IF  OP30_Gripper_RH_Gripper_ctrl.Axis_reference AND OP30_Gripper_RH_Open THEN
	OP30_Gripper_RH_Gripper_ctrl.Position:=OP30_Gripper_Wrk_POS;
	OP30_Gripper_RH_Gripper_ctrl.ABSmove_Start:=TRUE;
	IF OP30_Gripper_RH_Gripper_ctrl.pos_done AND In_range(OP30_Gripper_RH_Gripper_ctrl.Actual_Position,OP30_Gripper_Wrk_POS,1) THEN
		OP30_Gripper_RH_Open:=FALSE;
		OP30_Gripper_RH_Gripper_ctrl.ABSmove_Start:=0;
		OP30_Gripper_RH_State:=1;
	END_IF
END_IF

IF  OP30_Gripper_RH_Gripper_ctrl.Axis_reference AND OP30_Gripper_RH_Close THEN
	OP30_Gripper_RH_Gripper_ctrl.Position:=0;
	OP30_Gripper_RH_Gripper_ctrl.ABSmove_Start:=TRUE;
	IF OP30_Gripper_RH_Gripper_ctrl.pos_done AND In_range(OP30_Gripper_RH_Gripper_ctrl.Actual_Position,0.1,1) THEN
		OP30_Gripper_RH_Close:=FALSE;
		OP30_Gripper_RH_Gripper_ctrl.ABSmove_Start:=0;
		OP30_Gripper_RH_State:=0;
	END_IF	
END_IF

Test(IN:= OP30_Gripper_RH_State AND OP30_Gripper_LH_State , PT:=T#500MS);


OP30_GIUDE_GRP(														// FESTO GUIDE GRIPPER
	bAxis1_Ref_Switch:= , 
	bInit:=  , 
	bErrorReset:= Servo_Reset , 
	bEnable:= Servo_Enable , /// MACHINE ERR REGISTER CHANGE
	bMoveVelocity:= , 
	bHalt:= , 
	bManualMode:=OP30_ManualSelected AND MANUAL_SELECTED , 									//MANUAL REGISTER CHANGE
	fHomePos:= , 
	fOverride:= , 
	fTargetPosition:= OP30_GIUDE_GRP_ctrl.Position, 
	fTargetVelocity:= OP30_GIUDE_GRP_ctrl.Velocity, 
	fAcc:= , 
	fDec:= , 
	Servo_High_Limit:= 100,	
	Servo_Low_Limit:= -100,	 	
	WARNING_LIMIT:= 1,		
	Safe_move_Conditions:= Servo_Safety,
	TORQUE_APPLIED :=  , 					// CHANGE
	Axis:= SR30_GUIDE_GRP_AXIS, 
	bHome:= OP30_GIUDE_GRP_ctrl.Bsethome, 
	bSetPosition:= FESTO_NOT_NEED , 
	bMoveAbsolute:= OP30_GIUDE_GRP_ctrl.ABSmove_Start, 
	bMoveRelative:= NOT_REQ , 
	bMoveTorque:= NOT_REQ , 
	stManualModeAxis:= OP30_GIUDE_GRP_Manual_Axis, 
 	sAxisState=> OP30_GIUDE_GRP_ctrl.Axis_State, 
	baxis_in_home_pos=>OP30_GIUDE_GRP_ctrl.Axis_In_Home ,
	bAxis_ready=> , 
	bAxisInPosition=> , 
	bAxisError=> , 
	bAxisEnabled=> , 
	bAxisHomed=>, 
	bSetPositionDone=> , 
	bHaltDone=> , 
	bSTOPDone=> , 
	bHomeDone=>OP30_GIUDE_GRP_ctrl.Axis_Home_Done , 
	bDone=> , 
	bTorqueReached=> , 
	bsafe_to_move=> , 
	baxis_in_home_pos=> , 
	bABS_Pos_done=> OP30_GIUDE_GRP_ctrl.Axis_In_Pos, 
	Actual_position=>OP30_GIUDE_GRP_ctrl.Actual_Position,
	Actual_velocity=>OP30_GIUDE_GRP_ctrl.Actual_Velocity , 
	Actual_Torque=> );

END_PROGRAM

// ---- POUs/Programs/OP30/OP30_AUTOSEQUENCE.TcPOU
PROGRAM OP30_AUTOSEQUENCE
VAR
	OP30_Oring_OK 	: BOOL;
	FIXTURE_LH		: INT;
	FIXTURE_RH 		: INT;
	del : ton;
	tmp :BOOL;
	Jerk_Check	: TON;
	Gripper_Delay: TON;
	Gripper_Aft_Place_Delay	: TON;
	OP30_STN_MOVER: INT;
	Dry_run : BOOL;
	OP30_Cycle_Time_FB : FB_Cycletime;
	Guide_Control_Temp : BOOL;
	
	PAP_CYC_VAR : BOOL;
	OP30_PAP_Cycle_time : UDINT;
	OP30_Overall_Cyc_Time	: UDINT;
	OP30_PAP_Cycle_Time_FB : FB_Cycletime;
	OP30_Continous_Run : BOOL;
END_VAR

// AUTO MODE
IF (NOT OP30_AutoSelected OR  OP30_ErrorActive OR OP30_HomeRunning ) THEN
	OP30_AutoRunning:= FALSE;
	OP30_AutoSeq:= 10;
END_IF	

IF (NOT OP30_AutoSelected OR  OP30_ErrorActive ) THEN
	OP30_Conveyor_ON:=FALSE;
END_IF	

IF OP30_AutoSelected THEN
	OP30_GIUDE_GRP_ctrl.Position:=OP30_Guide_Pos;
	OP30_GIUDE_GRP_ctrl.Velocity:=50;
	SR30_Vert_servo_ctrl.Velocity:=OP30_HMI_Servo_Speed_Vertical;
	SR30_HORI_servo_ctrl.Velocity:=OP30_HMI_Servo_Speed_Horizontal;	
END_IF

IF NOT OP30_AutoRunning THEN
    OP30_GIUDE_GRP_ctrl.Position:=0;
	OP30_GIUDE_GRP_ctrl.Velocity:=50;
	IF NOT In_Range(OP30_GIUDE_GRP_ctrl.Actual_Position,0,1) THEN
		OP30_GIUDE_GRP_ctrl.ABSmove_Start:=TRUE;
	END_IF	
END_IF

CASE OP30_AutoSeq OF
	    10: IF (OP30_AutoSelected) THEN		// Check Automode Selected
				OP30_AutoSeq:=20;
	        END_IF
		
	    20:IF ( NOT OP30_ErrorActive) THEN		//Check No error
		       OP30_AutoSeq:=30;
      	   END_IF
		   
      	30:IF (NOT OP30_HomeRunning) THEN		//Check No Homerunning
      		   OP30_AutoSeq :=40;
      	   END_IF
		   
        40:IF (OP30_Main.OP30_Modeselection_FB.TempHomeOK)THEN	//Check Machine in Home
      		   OP30_AutoSeq:= 50;
      	   END_IF
		   
      	50:IF ( NOT OP30_OperationCompleted) THEN		// Check Operation Completed Reset
			   OP30_AutoSeq:=60;
      	   END_IF
		   
		60:IF  ( OP30_AutoRunning OR (NOT OP30_AutoRunning AND OP30_HMI_Cycle_Start )) THEN		//Machine Start in Fully Automatic or Press Cycle Start For Semi Automatic
		    OP30_GVL.OP30_HomeConditionOK:=TRUE;
	 			IF( OP30_Main.OP30_Modeselection_FB.HomeConditionOK AND OP30_AutoSelected) THEN
					OP30_GVL.OP30_AutoRunning:=TRUE;
					OP30_GVL.OP30_StepRunning:= FALSE;				
				ELSIF (OP30_Main.OP30_Modeselection_FB.HomeConditionOK AND OP30_StepSelected) THEN
					OP30_GVL.OP30_AutoRunning:=FALSE;
					OP30_GVL.OP30_StepRunning:= TRUE;
				END_IF;
		  END_IF
		   IF ((OP30_AutoRunning OR OP30_StepRunning) AND OP30_StartEnable) THEN
			   	OP30_GIUDE_GRP_ctrl.ABSmove_Start:=TRUE;
				OP30_Conveyor_ON:=TRUE;
				OP30_AutoSeq:= 65;
		   END_IF	
		   
		65 :  OP30_Gripper_LH_Close:=TRUE;  //CHECKING GRIPPER STATE BEFORE GRIPPING
			  OP30_Gripper_RH_Close:=TRUE;
			  IF NOT OP30_Gripper_LH_State AND NOT OP30_Gripper_RH_State THEN
				   OP30_AutoSeq:=66;
			  ELSE 	   
				   OP30_AutoSeq:=220;
			  END_IF 
		   
	    66: PAP_CYC_VAR:=1;
			IF OP30_pick_ready THEN
				OP30_AutoSeq:=70;
			ELSE 
				OP30_AutoSeq:=86;	
			END_IF 
			  
		70 : //MOVING HORIZONTAL SERVO TO PICK POSITION
			  IF (OP30_HORI_SERVO_ON_SFE_WRK OR OP30_HORI_SERVO_ON_HOME OR OP30_HORI_SERVO_ON_WRK_PLACE OR OP30_HORI_SERVO_ON_WRK_PICK )AND OP30_HORI_SERVO_POS_DONE AND NOT SR30_HORI_servo_ctrl.ABSmove_Start THEN 
			   SR30_Hori_servo_ctrl.Position:=OP30_HORI_SERVO_PICK_POS;
               OP30_AutoSeq:=80;
			  END_IF
			 
		80 :  SR30_HORI_servo_ctrl.ABSmove_Start := TRUE;     //HORIZONTAL SERVO MOVING
		       IF OP30_HORI_SERVO_ON_WRK_PICK THEN
				   SR30_HORI_servo_ctrl.ABSmove_Start := FALSE;
				   IF OP30_Gripper_LH_State AND OP30_Gripper_RH_State THEN
				        OP30_AutoSeq:=85;
				   ELSE 
						OP30_AutoSeq:=82;
				   END_IF
			   END_IF
		
	  	82 :  OP30_Gripper_LH_Close:=TRUE;  //CHECKING GRIPPER STATE BEFORE GRIPPING
			  OP30_Gripper_RH_Close:=TRUE;
			  IF NOT OP30_Gripper_LH_State AND NOT OP30_Gripper_RH_State THEN
				   OP30_AutoSeq:=85;
			  END_IF
			   
		85:	   // MOVING VERTICAL SERVO TO PICK POSITION
               IF  OP30_HORI_SERVO_ON_WRK_PICK AND (OP30_VERT_SERVO_ON_SFE_WRK OR OP30_VERT_SERVO_ON_HOME) AND OP30_VERT_SERVO_POS_DONE AND NOT SR30_VERT_servo_ctrl.ABSmove_Start   THEN
				   SR30_Vert_servo_ctrl.Position:=OP30_VERT_SERVO_PICK_POS;
				   SR30_VERT_servo_ctrl.ABSmove_Start := TRUE;
              	   OP30_AutoSeq:=100;			   
			   END_IF
			   
	    86:   IF (OP30_HORI_SERVO_ON_SFE_WRK OR OP30_HORI_SERVO_ON_HOME OR OP30_HORI_SERVO_ON_WRK_PLACE OR OP30_HORI_SERVO_ON_WRK_PICK )AND OP30_HORI_SERVO_POS_DONE AND NOT SR30_HORI_servo_ctrl.ABSmove_Start THEN 
			    SR30_Hori_servo_ctrl.Position:=OP30_HORI_SERVO_SAFE_PICK_POS;
			    SR30_HORI_servo_ctrl.ABSmove_Start := TRUE;
                OP30_AutoSeq:=90;
			  END_IF
  
		90 :   IF OP30_pick_ready THEN  // WAITING FOR O-RING TO BE OK AND THEN MOVING THE VERTICAL SERVO
			 		SR30_Hori_servo_ctrl.Position:=OP30_HORI_SERVO_PICK_POS;
					OP30_AutoSeq:=92;
		       END_IF
			   
		92:  SR30_Hori_servo_ctrl.ABSmove_Start := TRUE;
			 IF OP30_HORI_SERVO_ON_WRK_PICK THEN
				 SR30_Vert_servo_ctrl.Position:=OP30_VERT_SERVO_PICK_POS;
				 SR30_VERT_servo_ctrl.ABSmove_Start := TRUE;
				 OP30_AutoSeq:=100;
			 END_IF
						  						   			   
	   100 : IF OP30_VERT_SERVO_ON_WRK_PICK AND NOT SR30_VERT_servo_ctrl.ABSmove_Start THEN
				 SR30_VERT_servo_ctrl.ABSmove_Start := FALSE;
				 SR30_Vert_servo_ctrl.Position:=OP30_VERT_SERVO_SFE_WRK_POS; // FEEDING SAFE-WORK POSITION TO VERTICAL SERVO
              	 OP30_AutoSeq:=110;			    				   
			 END_IF	   
			   
       110:	IF NOT OP30_Grip_LH_Bypass THEN
				OP30_Gripper_LH_Open:=TRUE; 
			END_IF	
			IF NOT OP30_Grip_RH_Bypass THEN
    			OP30_Gripper_RH_Open:=TRUE;
			END_IF	
			IF Gripper_Delay.Q THEN
				 OP30_AutoSeq:=120;
		    END_IF 
    		
       120: SR30_Hori_servo_ctrl.Position:=(OP30_HORI_SERVO_PICK_POS+OP30_Hori_Ser_Jerk_Pos);
	   		SR30_HORI_servo_ctrl.ABSmove_Start := 1;
			IF Jerk_Check.Q THEN
				OP30_AutoSeq:=130;
			END_IF    
    		   
       130: SR30_VERT_servo_ctrl.ABSmove_Start := TRUE;	   //MOVING VERTICL SERVO TO SAFE-WORK
            IF OP30_VERT_SERVO_ON_SFE_WRK  THEN
    	      SR30_VERT_servo_ctrl.ABSmove_Start := FALSE;
			  OP30_pick_done:=TRUE;
              OP30_AutoSeq:=140;   
    		END_IF
    		   
       140: IF (NOT OP30_Gripper_LH_State AND OP30_Grip_LH_Bypass ) AND OP30_Gripper_RH_State THEN  
    			OP30_AutoSeq:=150;
			ELSIF (NOT OP30_Gripper_RH_State AND OP30_Grip_RH_Bypass) AND OP30_Gripper_LH_State THEN
				OP30_AutoSeq:=150;
			ELSIF OP30_Gripper_LH_State AND OP30_Gripper_RH_State THEN  
    			OP30_AutoSeq:=150;
			ELSIF (NOT OP30_Gripper_LH_State AND NOT OP30_Grip_LH_Bypass) OR (NOT OP30_Gripper_RH_State AND NOT OP30_Grip_RH_Bypass) THEN	
				OP30_AutoSeq:=220;
			ELSIF OP30_Grip_LH_Bypass AND OP30_Grip_RH_Bypass THEN
				OP30_AutoSeq:=250;
			END_IF
    	    		  
       150:  IF OP30_VERT_SERVO_ON_SFE_WRK  THEN // FEEDING PLACE POSITION TO HORIZONTAL SERVO
    		   SR30_Hori_servo_ctrl.Position:=OP30_HORI_SERVO_PLACE_POS;
              OP30_AutoSeq:=160;			 
    		 END_IF
    		   
       160:  SR30_HORI_servo_ctrl.ABSmove_Start := TRUE;    // MOVING HORIZONTAL SERVO TO PLACE POSITION
    		   IF OP30_HORI_SERVO_ON_WRK_PLACE THEN
    			 SR30_HORI_servo_ctrl.ABSmove_Start := FALSE;
    			 OP30_AutoSeq:=170;
    		   END_IF
       
       170: PAP_CYC_VAR:=0;
			IF OP30_HORI_SERVO_ON_WRK_PLACE AND NOT SR30_VERT_servo_ctrl.ABSmove_Start AND OP30_VERT_SERVO_ON_SFE_WRK AND OP30_STN_ENABLE THEN
    	   		SR30_Vert_servo_ctrl.Position:=OP30_VERT_SERVO_PLACE_POS;
              	OP30_AutoSeq:=175;		
      		END_IF
			
	   175: IF FIXTURE_LH<>20 AND FIXTURE_RH<>20 THEN
		   		OP30_AutoSeq:=250;	
			ELSIF FIXTURE_LH<>20 OR FIXTURE_RH<>20 THEN
				OP30_AutoSeq:=260;	
			ELSE
				OP30_AutoSeq:=180;		
	  	    END_IF
    		
       180: SR30_Vert_servo_ctrl.Position:=OP30_VERT_SERVO_PLACE_POS;
			SR30_VERT_servo_ctrl.ABSmove_Start := TRUE; //MOVING VERTICAL SERVO TO PLACE POSITION
    		IF OP30_VERT_SERVO_ON_WRK_PLACE THEN
    			SR30_VERT_servo_ctrl.ABSmove_Start := FALSE;
    		    OP30_AutoSeq:=190;					
    		END_IF	
			
       190: IF FIXTURE_LH=20 AND NOT OP30_Grip_LH_Bypass THEN 
				OP30_Gripper_LH_Close:=TRUE;	
			END_IF	
			IF FIXTURE_RH=20 AND NOT OP30_Grip_RH_Bypass THEN 
				OP30_Gripper_RH_Close:=TRUE;
			END_IF			
			OP30_AutoSeq	:=200;
			OP30_CURR_MOVER	:= OP30_STN_MOVER;
				
	
       200:  //MOVING BACK TO VERTICAL SERVO SAFE POSITION
    		 IF OP30_VERT_SERVO_ON_WRK_PLACE AND NOT SR30_VERT_servo_ctrl.ABSmove_Start THEN
    		   SR30_Vert_servo_ctrl.Position:=OP30_VERT_SERVO_SFE_WRK_POS;
			   IF Gripper_Aft_Place_Delay.Q THEN
                OP30_AutoSeq:=201;
			   END_IF			   
    		 END_IF 
    		 
	   201: IF Dry_Run THEN
				OP30_AutoSeq:=210; 
			END_IF
			IF  FIXTURE_LH=20 AND FIXTURE_RH=20 THEN
				MOVER_CMP_STATUS[OP30_CURR_MOVER][1]:=30 ;
				MOVER_CMP_STATUS[OP30_CURR_MOVER][2]:=30 ;
				OP30_AutoSeq:=210;
			ELSIF FIXTURE_LH=20 THEN
				MOVER_CMP_STATUS[OP30_CURR_MOVER][1]:=30 ;
				OP30_AutoSeq:=210;
			ELSIF FIXTURE_RH=20 THEN
				MOVER_CMP_STATUS[OP30_CURR_MOVER][2]:=30 ;
				OP30_AutoSeq:=210;
			END_IF		 
			 
       210:	   //PROCEEDING FOR NEXT CYCLE 
			  SR30_VERT_servo_ctrl.ABSmove_Start := TRUE;         
              IF OP30_VERT_SERVO_ON_SFE_WRK OR OP30_VERT_SERVO_ON_HOME  THEN
    			SR30_VERT_servo_ctrl.ABSmove_Start := FALSE;			  
				OP30_STN_ENABLE:=0;
				IF OP30_Gripper_LH_State OR OP30_Gripper_RH_State THEN
					OP30_AutoSeq:=220;
				ELSIF (MOVER_CMP_STATUS[OP30_STN_MOVER][1]=30 OR MOVER_CMP_STATUS[OP30_STN_MOVER][2]=30) OR Dry_Run THEN
					STATION_DONE[OP30_CURR_MOVER][OP30_XTS_POS_NO]	:= TRUE;
					IF MOVER_STP_NO[OP30_CURR_MOVER]<>((OP30_XTS_POS_NO*10)+1)THEN
						OP30_AutoSeq:=66;  
					END_IF	
    		  	END_IF  			  
			  END_IF
    		  
       220:  IF (OP30_VERT_SERVO_ON_SFE_WRK OR OP30_VERT_SERVO_ON_HOME OR OP30_VERT_SERVO_ON_WRK_PLACE OR OP30_VERT_SERVO_ON_WRK_PICK) AND NOT SR30_HORI_servo_ctrl.ABSmove_Start AND (OP30_HORI_SERVO_ON_WRK_PLACE OR OP30_HORI_SERVO_ON_WRK_Pick)  THEN
    		   SR30_Hori_servo_ctrl.Position:=OP30_HORI_SERVO_SFE_WRK_POS;
			   SR30_Vert_servo_ctrl.Position:=OP30_VERT_SERVO_SFE_WRK_POS;
               OP30_AutoSeq:=240;			  
    		 END_IF  
    	
       240: SR30_VERT_servo_ctrl.ABSmove_Start := TRUE;	
			IF OP30_VERT_SERVO_ON_SFE_WRK THEN
			 	SR30_HORI_servo_ctrl.ABSmove_Start := TRUE;
             	IF OP30_HORI_SERVO_ON_SFE_WRK THEN
    	  	 	  SR30_HORI_servo_ctrl.ABSmove_Start := FALSE;
      		 	  OP30_Gripper_RH_Close:=TRUE;	
    		 	  OP30_Gripper_LH_Close:=TRUE; 			   
      		 	END_IF
			END_IF	
    		IF NOT OP30_Gripper_LH_State AND NOT OP30_Gripper_RH_State THEN
    		   OP30_AutoSeq:=66;
    		END_IF
			 		
		250://MOVER_CMP_STATUS[OP30_CURR_MOVER][1]:=31;
			//MOVER_CMP_STATUS[OP30_CURR_MOVER][2]:=31;
			OP30_STN_ENABLE:=0;
			IF 	(MOVER_CMP_STATUS[OP30_STN_MOVER][1]=31 AND MOVER_CMP_STATUS[OP30_STN_MOVER][2]=31) THEN
				MOVER_STP_NO[OP30_CURR_MOVER]	:= (OP160_XTS_POS_NO*10);
			ELSE		
				STATION_DONE[OP30_CURR_MOVER][OP30_XTS_POS_NO]	:= TRUE;
			END_IF	
			IF MOVER_STP_NO[OP30_CURR_MOVER]<>((OP30_XTS_POS_NO*10)+1)THEN 
				OP30_CURR_MOVER	:= 0;
				OP30_AutoSeq	:=170;  
			END_IF

	   260: SR30_Hori_servo_ctrl.Position:=OP30_HORI_SERVO_SFE_WRK_POS;
			SR30_Hori_servo_ctrl.ABSmove_Start:=TRUE;
			IF OP30_HORI_SERVO_ON_SFE_WRK THEN
				OP30_AutoSeq:=270; 
			END_IF
			
	   270: IF FIXTURE_LH<>20 AND NOT OP30_Grip_LH_Bypass THEN
				OP30_Gripper_LH_Close:=TRUE;
				IF NOT OP30_Gripper_LH_State THEN
					OP30_AutoSeq:=280; 
				END_IF
			ELSE
				OP30_AutoSeq:=280;	
			END_IF	
			
	   280: IF FIXTURE_RH<>20 AND NOT OP30_Grip_RH_Bypass THEN
				OP30_Gripper_RH_Close:=TRUE;
				IF NOT OP30_Gripper_RH_State THEN
					OP30_AutoSeq:=290; 
				END_IF
			ELSE
				OP30_AutoSeq:=290;	
			END_IF	

	   290: SR30_Hori_servo_ctrl.Position:=OP30_HORI_SERVO_PLACE_POS;
			SR30_Hori_servo_ctrl.ABSmove_Start:=TRUE;
			IF OP30_HORI_SERVO_ON_WRK_PLACE THEN
				OP30_AutoSeq:=180;	
			END_IF
					
      300: IF (OP30_HORI_SERVO_ON_SFE_WRK OR OP30_HORI_SERVO_ON_HOME OR OP30_HORI_SERVO_ON_SFE_WRK_PICK ) AND NOT SR30_HORI_servo_ctrl.ABSmove_Start AND OP30_Size_Rej THEN
		  		SR30_Hori_servo_ctrl.Position:=OP30_HORI_SERVO_PICK_POS;	
				OP30_Size_Rej:=0;		
				OP30_AutoSeq:=310;
	       END_IF
		   
	  310: SR30_Hori_servo_ctrl.ABSmove_Start  := TRUE;
		   IF OP30_HORI_SERVO_ON_WRK_PICK THEN
		  		SR30_Vert_servo_ctrl.Position:=OP30_VERT_SERVO_PICK_POS;
				OP30_AutoSeq:=320;
	  	   END_IF
		   
	 320: SR30_VERT_servo_ctrl.ABSmove_Start := TRUE;
		  IF OP30_VERT_SERVO_ON_WRK_PICK THEN
		 	  OP30_Gripper_LH_Open:=OP30_LH_Size_NOK;
			  OP30_Gripper_RH_Open:=OP30_LH_Size_NOK;
			  OP30_Size_Rej_Complete:=1;
			  OP30_AutoSeq:=220;
	 	  END_IF
  
	   
END_CASE

IF OP30_Size_Rej THEN
	OP30_AutoSeq:=300;
END_IF

Dry_Run:=All_Station_Dry_Run;
IF Dry_run THEN
	FIXTURE_LH :=20;	
    FIXTURE_RH :=20;
ELSE 
	FIXTURE_LH:=MOVER_CMP_STATUS[OP30_STN_MOVER][1];
	FIXTURE_RH:=MOVER_CMP_STATUS[OP30_STN_MOVER][2];	
END_IF

OP30_Cycle_Time_FB(i_b_startTime:=OP30_STN_ENABLE , i_b_stopTime:= NOT OP30_STN_ENABLE , o_t_StationTime=>OP30_Cycle_time );					
OP30_PAP_Cycle_Time_FB(i_b_startTime:=PAP_CYC_VAR , i_b_stopTime:= NOT PAP_CYC_VAR , o_t_StationTime=>OP30_PAP_Cycle_time );					
OP30_Overall_Cyc_Time:=OP30_Cycle_time+OP30_PAP_Cycle_time;

Gripper_Delay(IN:=(OP30_AutoSeq=110),PT:=T#700MS);
Gripper_Aft_Place_Delay(IN:=(OP30_AutoSeq=200),PT:=T#700MS);
Jerk_Check(IN:= OP30_AutoSeq=120 , PT:=T#100MS);


del(IN:=tmp,PT:=T#700MS);
IF del.Q THEN
	tmp:=FALSE;
END_IF

OP30_STN_ENABLE:=OP30_Continous_Run;
//######################## 				ENABLE CONDTION   				#################


	OP30_STN_MOVER	:= MOVER_POSITION[OP30_XTS_POS_NO];
	
IF AUTO_WITH_XTS THEN
IF OP30_STN_MOVER>0 THEN
IF NOT(END_OF_CYCLE AND MOVER_CMP_STATUS[OP30_STN_MOVER][1]=5 AND MOVER_CMP_STATUS[OP30_STN_MOVER][2]=5)THEN	
OP30_STN_ENABLE	:= MOVER_POS_RECHED[OP30_STN_MOVER] AND ((MOVER_CMP_STATUS[OP30_STN_MOVER][1]=20)OR 
					(MOVER_CMP_STATUS[OP30_STN_MOVER][2]=20)) AND STATION_ENABLE_CONTROL;
ELSE
	STATION_DONE[OP30_STN_MOVER][OP30_XTS_POS_NO]			:= TRUE;	
END_IF
ELSE
OP30_STN_ENABLE				:= FALSE;	
END_IF	
END_IF

END_PROGRAM

// ---- POUs/Programs/OP30/OP30_Conveyor_Cam_Seq.TcPOU
PROGRAM OP30_Conveyor_Cam_Seq
VAR
	Conv_Cam_Step : INT;
	LH_Cam_OK	  : BOOL;
	RH_Cam_OK	  : BOOL;
	LH_Pic		  : R_TRIG;
	RH_Pic		  : R_TRIG;	
	Conv_Step_no  : INT;
	OP30_Conveyor_FB : Servo_Conveyor_FB;
	Conveyor_Track_Delay	: TON;
	Conveyor_Track_OFF_Delay	: TON;
	B1 : BOOL;
	B2 : BOOL;
	B3 : BOOL;
	B4 : BOOL;	
	B5 : BOOL;
	B6 : BOOL;
	Conveyor_Velocity_mode	: BOOL;
	Conveyor_Conti_run		: BOOL;
	OP30_Miss_Trigger: BOOL;
	Temp_Counter_LH: UINT;
	Temp_Counter_RH: UINT;
	OP30_Camera_Trigger_Ack: BOOL;
	Temp: BOOL;
	Toggle_Pos_LH : R_TRIG;
	Toggle_Neg_LH : F_TRIG;
	Toggle_Pos_RH : R_TRIG;
	Toggle_Neg_RH : F_TRIG;
	LH_Cam_Completed : BOOL;
	RH_Cam_Completed : BOOL;
	Drum_Jam_Timer	 : TON;
	OP30_Camera_Bypass : BOOL;
	Control : BOOL;
END_VAR


Toggle_Pos_LH(CLK:=OP30_Camera_FB.OP30_LH_Inspection_Status.Inspection_Completed);
Toggle_Neg_LH(CLK:=OP30_Camera_FB.OP30_LH_Inspection_Status.Inspection_Completed);
Toggle_Pos_RH(CLK:=OP30_Camera_FB.OP30_RH_Inspection_Status.Inspection_Completed);
Toggle_Neg_RH(CLK:=OP30_Camera_FB.OP30_RH_Inspection_Status.Inspection_Completed);

IF Toggle_Pos_LH.Q OR Toggle_Neg_LH.Q THEN
	LH_Cam_Completed:=1;	
END_IF
IF Toggle_Pos_RH.Q OR Toggle_Neg_RH.Q THEN
	RH_Cam_Completed:=1;	
END_IF


IF MANUAL_SELECTED AND OP30_ManualSelected THEN               
	IF I30_DRUM_CONV_REV_I304_3 THEN
		SR30_Conv_servo_status.targetVelocity:=OP30_Conv_Rev_Speed_6_3;
		SR30_Conv_servo_status.moveVelocity:=I30_DRUM_CONV_REV_I304_3;
 	ELSIF I30_DRUM_CONV_FWD_I304_4 THEN
		SR30_Conv_servo_status.targetVelocity:=OP30_Conv_Fwd_Speed_7_89;
		SR30_Conv_servo_status.moveVelocity:=I30_DRUM_CONV_FWD_I304_4;	
	ELSE 	
		SR30_Conv_servo_status.moveVelocity:=0;   	
	END_IF  	
END_IF   

IF (NOT OP30_AutoRunning OR (NOT OP30_LH_Camera_Online OR NOT OP30_RH_Camera_Online)) AND NOT OP30_Camera_Bypass THEN
	Conv_Cam_Step:=10;
END_IF  

CASE Conv_Cam_Step OF
	10: 	OP30_LH_Camera_OK :=0;
            OP30_LH_Camera_NOK:=0;
	        OP30_RH_Camera_OK :=0;
	        OP30_RH_Camera_NOK:=0;	
			LH_Cam_Completed  :=0;
			RH_Cam_Completed  :=0;		
			OP30_Camera_Done  :=0;
			OP30_LH_Clr_OK 	  :=0;
		    OP30_RH_Clr_OK 	  :=0;		
			OP30_LH_Size_OK	  :=0;
		    OP30_RH_Size_OK	  :=0;	
			Conv_Cam_Step	  :=11;	
	
	11: IF ((OP30_Camera_Trigger AND (NOT OP30_Camera_Done)) OR OP30_Miss_Trigger ) AND NOT OP30_Camera_Bypass THEN
			OP30_LH_Camera_Trigger:=1;
			OP30_RH_Camera_Trigger:=1;
			Conv_Cam_Step		  :=15;	
		END_IF

	15:	IF LH_Cam_Completed AND RH_Cam_Completed THEN
			OP30_LH_Camera_Trigger:=0;
			OP30_RH_Camera_Trigger:=0;
			OP30_Camera_Trigger :=0;
			OP30_Miss_Trigger	:=0;
			Conv_Cam_Step:=25;
		END_IF  
	   
	25: IF OP30_Camera_FB.OP30_LH_Cam_Result[0]=1 AND OP30_Camera_FB.OP30_RH_Cam_Result[0]=1 THEN
			OP30_LH_Camera_OK:=1;
			OP30_RH_Camera_OK:=1;
			Conv_Cam_Step    :=50;
		ELSIF (OP30_Camera_FB.OP30_LH_Cam_Result[2]<>1 OR OP30_Camera_FB.OP30_RH_Cam_Result[2]<>1) THEN	
			OP30_One_Cycle  :=1;
			Conv_Cam_Step   :=50;
		ELSIF (OP30_Camera_FB.OP30_LH_Cam_Result[1]=1 OR OP30_Camera_FB.OP30_RH_Cam_Result[1]=1) AND (OP30_Camera_FB.OP30_LH_Cam_Result[2]=1 AND OP30_Camera_FB.OP30_RH_Cam_Result[2]=1) THEN			
			IF OP30_Camera_FB.OP30_LH_Cam_Result[0]=1 THEN
				OP30_LH_Camera_OK:=1;
			END_IF
			IF OP30_Camera_FB.OP30_RH_Cam_Result[0]=1 THEN
				OP30_RH_Camera_OK:=1;
			END_IF
			Conv_Cam_Step:=30;
		END_IF	
			
   30: 	IF OP30_Camera_FB.OP30_LH_Cam_Result[1]=1 THEN
	   		OP30_LH_Camera_NOK:=1;
  	    END_IF
		IF OP30_Camera_FB.OP30_RH_Cam_Result[1]=1 THEN
	   		OP30_RH_Camera_NOK:=1;
  	    END_IF
		Conv_Cam_Step:=50;
		
   50:  OP30_Camera_Done:=1;
   		Temp_Counter_LH:=OP30_Camera_FB.OP30_LH_Acquisition_ID;
		Temp_Counter_RH:=OP30_Camera_FB.OP30_RH_Acquisition_ID;
		IF Conv_Step_no>75 THEN
			Conv_Cam_Step   :=10;
			OP30_Camera_Done:=0;
		END_IF
   	    
END_CASE


IF OP30_Model='6.3' THEN
	OP30_Conv_Fwd_Time:=OP30_Conv_Fwd_Time_6_3;
	OP30_Conv_Rev_Time:=OP30_Conv_Rev_Time_6_3;
	OP30_Conveyor_FWD_Speed:= OP30_Conv_Fwd_Speed_6_3;
	OP30_Conveyor_REV_Speed:= OP30_Conv_Rev_Speed_6_3;
END_IF

IF OP30_Model='7.89' THEN
	OP30_Conv_Fwd_Time:=OP30_Conv_Fwd_Time_7_89;
	OP30_Conv_Rev_Time:=OP30_Conv_Rev_Time_7_89;
	OP30_Conveyor_FWD_Speed:= OP30_Conv_Fwd_Speed_7_89;
	OP30_Conveyor_REV_Speed:= OP30_Conv_Rev_Speed_7_89;
END_IF

Conveyor_Velocity_mode:=1;

OP30_Conveyor_FB(
	Conveyor_Prgrm_Start:= OP30_Conveyor_ON AND OP30_AutoRunning, 
	Conveyor_Prgrm_Reset:= , 
	Conveyor_Continuous_Run:= Conveyor_Conti_run,
	Conveyor_FWD_Position	:= OP30_Conv_Fwd_Pos,
    Conveyor_REV_Position	:= OP30_Conv_Rev_Pos,
    Velocity_mode			:= Conveyor_Velocity_mode,
	Camera_Trigger_OK := OP30_Camera_Done OR OP30_Camera_Bypass ,
	Fwd_Time_IP:= OP30_Conv_Fwd_Time, 
	Rev_Time_IP:= OP30_Conv_Rev_Time, 
	Conveyor_FWD_Speed:=OP30_Conveyor_FWD_Speed , 
	Conveyor_REV_Speed:=OP30_Conveyor_REV_Speed , 
	LH_Work_Sensor:=CR30_LH_Rej_Cyl.Sensor2 , 
	LH_Home_Sensor:=CR30_LH_Rej_Cyl.Sensor1 , 
	RH_Work_Sensor:=CR30_RH_Rej_Cyl.Sensor2 , 
	RH_Home_Sensor:=CR30_RH_Rej_Cyl.Sensor1 ,
	Track_Overflow := Conveyor_Track_OFF_Delay.Q,
	Track_Sensor_FB := Conveyor_Track_Delay.Q, 
	LH_Camera_OK  :=  OP30_LH_Camera_OK OR OP30_Camera_Bypass, 
	LH_Camera_NOK := OP30_LH_Camera_NOK, 
	RH_Camera_OK  :=  OP30_RH_Camera_OK OR OP30_Camera_Bypass, 
	RH_Camera_NOK := OP30_RH_Camera_NOK,
	Drum_ON=> O30_DRUM_MTR_FWD_Q304_4, 
	Camera_Trigger_Ack=> OP30_Camera_Trigger_Ack,
	Camera_trigger := OP30_Camera_Trigger , 
	LH_Work_Coil=>CR30_LH_Rej_Cyl_wrk , 
	LH_Home_Coil=>CR30_LH_Rej_Cyl_hme , 
	RH_Work_Coil=>CR30_RH_Rej_Cyl_wrk,
	RH_Home_Coil=>CR30_RH_Rej_Cyl_hme,
	Ready_to_Pick=> OP30_pick_ready , 
	Step_Num => Conv_Step_no,
	Pick_Done       :=  OP30_pick_done , 
	One_Cycle		:=  OP30_One_Cycle,
	Conveyor_Servo_Control_Structure:= SR30_CONV_servo_ctrl );

Conveyor_Track_Delay(IN:= NOT I30_DRUM_FEED_CONV1_OVERFLW_I1100_0 OR NOT I30_DRUM_FEED_CONV2_OVERFLW_I1100_1,PT:=INT_TO_TIME(OP30_Drum_ON_Time));	
Conveyor_Track_OFF_Delay(IN:=I30_DRUM_FEED_CONV1_OVERFLW_I1100_0 AND I30_DRUM_FEED_CONV2_OVERFLW_I1100_1,    PT:=INT_TO_TIME(OP30_Drum_OFF_Time));   
	
IF 	OP30_AutoRunning THEN
	IF Conveyor_Track_OFF_Delay.Q THEN
		O30_DRUM_MTR_FWD_Q304_4:=0;
	END_IF
	//IF Conveyor_Track_Delay.Q THEN
	//	O30_DRUM_MTR_FWD_Q304_4:=1;
	//END_IF
	O30_AIR_PURGE_ON_Q1153_2:=1;
	O30_DRUM_RUN_IND_Q305_0:=O30_DRUM_MTR_FWD_Q304_4;
ELSE
	//SR30_CONV_servo_ctrl.VELmove_Start:=0;
	O30_DRUM_MTR_FWD_Q304_4:=I30_DRUM_OFF_ON_I304_2;
    O30_DRUM_RUN_IND_Q305_0:=I30_DRUM_OFF_ON_I304_2;
    O30_AIR_PURGE_ON_Q1153_2 :=I30_DRUM_OFF_ON_I304_2;
END_IF

//O30_DRUM_MTR_FWD_Q304_4:=I30_DRUM_OFF_ON_I304_2;

IF OP30_AutoRunning AND Control THEN
	Drum_Jam_Timer(IN:=(NOT I30_DRUM_FEED_CONV1_OVERFLW_I1100_0)OR(NOT I30_DRUM_FEED_CONV2_OVERFLW_I1100_1)); 
	Drum_Jam_Timer(PT:=T#40S);
	IF Drum_Jam_Timer.Q THEN
		OP30_ErrorActive:=1;
	END_IF
END_IF

LH_Pic(CLK:=OP30_LH_Picture_Taken);
IF LH_Pic.Q THEN
	LH_Cam_OK:=1;
END_IF

RH_Pic(CLK:=OP30_RH_Picture_Taken);
IF RH_Pic.Q THEN
	RH_Cam_OK:=1;
END_IF

END_PROGRAM

// ---- POUs/Programs/OP30/OP30_Camera_FB.TcPOU
PROGRAM OP30_Camera_FB
VAR
	OP30_LH_Camera 			             :  FB_Cognex_ProfiNET_1;
	OP30_LH_Acquisition_Status   AT %I*  :	Acquisition_Status;
	OP30_LH_Inspection_Status    AT %I*  :	Inspection_Status;	
	OP30_LH_Acquisition_ID       AT %I*  :	UINT;
	OP30_LH_Inspection_ID   	 AT %I*  :	UINT;
	OP30_LH_Error_code      	 AT %I*  :	UINT;
	OP30_LH_Current_Job_ID  	 AT %I*  :	UINT;
	OP30_LH_Result_code     	 AT %I*  :	UINT;
	OP30_LH_Cam_Result      	 AT %I*  :	ARRAY[0..63] OF BYTE;
	OP30_LH_Acquisition_Control AT %Q*   :   Acquisition_Control;
	OP30_LH_Inspection_Control  AT %Q*   :   Inspection_Control;
	OP30_LH_Command_word		AT %Q*   :   UINT;
	OP30_LH_Union                        :   UNION_64Byte;
	
	OP30_RH_Camera 			             :   FB_Cognex_ProfiNET_1;	
	OP30_RH_Acquisition_Status AT %I*    :	Acquisition_Status;
	OP30_RH_Inspection_Status  AT %I*    :	Inspection_Status;	
	OP30_RH_Acquisition_ID     AT %I*    :	UINT;
	OP30_RH_Inspection_ID   	 AT %I*  :	UINT;
	OP30_RH_Error_code      	 AT %I*  :	UINT;
	OP30_RH_Current_Job_ID  	 AT %I*  :	UINT;
	OP30_RH_Result_code     	 AT %I*  :	UINT;
	OP30_RH_Cam_Result      	 AT %I*  :	ARRAY[0..63] OF BYTE;
	OP30_RH_Acquisition_Control AT %Q*   :  Acquisition_Control;
	OP30_RH_Inspection_Control  AT %Q*   :  Inspection_Control;
	OP30_RH_Command_word		AT %Q*   :  UINT;
	OP30_RH_Union                        :  UNION_64Byte;
END_VAR

OP30_LH_Camera (
	tTimeout:= , 
	sJob_Name:= , 
	camera_ready=> OP30_LH_Camera_Ready,
	Camera_online=> OP30_LH_Camera_Online,
	stCognex_record_status:=OP30_LH_Acquisition_Status, 
	Acquisition_ID:=OP30_LH_Acquisition_ID , 
	stCognex_Inspection_status:=OP30_LH_Inspection_Status, 
	Error_Code:=OP30_LH_Error_code , 
	wcommand_control_in:= OP30_LH_Current_Job_ID, 
	aResults_64_Bytes:= OP30_LH_Cam_Result, 
	number_of_inspections:=OP30_LH_Inspection_ID , 
	iresult_code:= OP30_LH_Result_code, 
	bTarget_job_ID:=OP30_LH_Target_Job_ID , 
	Error_Status_message=> OP30_LH_Error_status, 
	bError=> OP30_LH_Camera_Error, 
	stCognex_record_control=>OP30_LH_Acquisition_Control , 
	stCognex_inspection_control=>OP30_LH_Inspection_Control , 
	wCommandControl_out=>OP30_LH_Command_word , 
	aUser_data_64_Byte=> OP30_LH_Union.aArrayOfByte, 
	bJob_loading_completed=>OP30_LH_Job_Change_Complete , 
	bJob_load_failed=>OP30_LH_Job_Change_Error , 
	bInspection_Result_IO=>  , 
	bInspection_Result_NIO=> , 
	bTXTSM_Error_Job_Change=> OP30_LH_Job_Change_Error, 
	bPictureTakenComplete=> OP30_LH_Picture_Taken, 
	Loaded_Job_ID=>OP30_LH_Loaded_Job_ID	 , 
	bClear_Error:= HMI_Reset, 
	bJob_change_start:= OP30_LH_Camera_Job_Change_start, 
	TXTSM_camera_not_online=>OP30_LH_Camera_Error	 , 
	bTrigger_start:= OP30_LH_Camera_Trigger );

OP30_RH_Camera (
	tTimeout:= , 
	sJob_Name:= , 
	camera_ready=> OP30_RH_Camera_Ready,
	Camera_online=> OP30_RH_Camera_Online,
	stCognex_record_status:=OP30_RH_Acquisition_Status, 
	Acquisition_ID:=OP30_RH_Acquisition_ID , 
	stCognex_Inspection_status:=OP30_RH_Inspection_Status, 
	Error_Code:=OP30_RH_Error_code , 
	wcommand_control_in:= OP30_RH_Current_Job_ID, 
	aResults_64_Bytes:= OP30_RH_Cam_Result, 
	number_of_inspections:=OP30_RH_Inspection_ID , 
	iresult_code:= OP30_RH_Result_code, 
	bTarget_job_ID:=OP30_RH_Target_Job_ID , 
	Error_Status_message=> OP30_RH_Error_status, 
	bError=> OP30_RH_Camera_Error, 
	stCognex_record_control=>OP30_RH_Acquisition_Control , 
	stCognex_inspection_control=>OP30_RH_Inspection_Control , 
	wCommandControl_out=>OP30_RH_Command_word , 
	aUser_data_64_Byte=> OP30_RH_Union.aArrayOfByte, 
	bJob_loading_completed=>OP30_RH_Job_Change_Complete , 
	bJob_load_failed=>OP30_RH_Job_Change_Error , 
	bInspection_Result_IO=>  , 
	bInspection_Result_NIO=> , 
	bTXTSM_Error_Job_Change=> OP30_RH_Job_Change_Error, 
	bPictureTakenComplete=> OP30_RH_Picture_Taken, 
	Loaded_Job_ID=>OP30_RH_Loaded_Job_ID	 , 
	bClear_Error:= HMI_Reset, 
	bJob_change_start:= OP30_RH_Camera_Job_Change_start, 
	TXTSM_camera_not_online=>OP30_RH_Camera_Error	 , 
	bTrigger_start:= OP30_RH_Camera_Trigger );

END_PROGRAM

// ---- POUs/Programs/OP30/OP30_Error.TcPOU
PROGRAM OP30_Error
VAR
	OP30_Step_Err_1: TON;
	OP30_Step_Err_2: TON;
	OP30_Step_Err_3: TON;
	OP30_Step_Err_4: TON;
	OP30_Step_Err_5: TON;
	OP30_Step_Err_6: TON;
END_VAR


// Set ERROR ACTIVE
IF ((OP30_GVL.OP30_ErrorWord_0<>0) OR (OP30_GVL.OP30_ErrorWord_1<>0) OR (OP30_GVL.OP30_ErrorWord_2<>0)) THEN
	OP30_GVL.OP30_ErrorActive:= TRUE;
END_IF

//Reset ErrorActive
IF (OP30_GVL.OP30_HMI_Reset OR HMI_Reset) THEN 
	OP30_GVL.OP30_ErrorActive:= FALSE;
	OP30_GVL.OP30_ErrorWord_0:= 0;
	OP30_GVL.OP30_ErrorWord_1:= 0;
	OP30_GVL.OP30_ErrorWord_2:= 0;	
END_IF

// Auto Seq Step Error

//Horizontal Servo is not in home or safe-work position 
OP30_Step_Err_1(IN:=(OP30_GVL.OP30_AutoSeq=70) , PT:=T#5S , Q=> , ET=> );
IF (OP30_GVL.OP30_AutoSeq=70 AND OP30_Step_Err_1.Q) THEN
	OP30_GVL.OP30_ErrorWord_0.0:=TRUE;
END_IF


//Horizontal Servo not reaching pick position 
OP30_Step_Err_1(IN:=(OP30_GVL.OP30_AutoSeq=80) , PT:=T#5S , Q=> , ET=> );
IF (OP30_GVL.OP30_AutoSeq=80 AND NOT OP30_HORI_SERVO_ON_WRK_PICK AND OP30_Step_Err_1.Q) THEN
	OP30_GVL.OP30_ErrorWord_0.1:=TRUE;
END_IF

// Gripper is not closing
OP30_Step_Err_2(IN:=OP30_GVL.OP30_AutoSeq=82 , PT:=T#5S , Q=> , ET=> );
IF (OP30_GVL.OP30_AutoSeq=82 AND OP30_Step_Err_2.Q) THEN
	OP30_GVL.OP30_ErrorWord_0.2:=TRUE;
END_IF

// Vertical Servo not reaching work position 
OP30_Step_Err_3(IN:=OP30_GVL.OP30_AutoSeq=100 , PT:=T#5S , Q=> , ET=> );
IF (OP30_GVL.OP30_AutoSeq=100 AND OP30_Step_Err_3.Q) THEN
	OP30_GVL.OP30_ErrorWord_0.3:=TRUE;
END_IF

// Vertical Servo not reaching safe-work position 
OP30_Step_Err_3(IN:=OP30_GVL.OP30_AutoSeq=130 , PT:=T#5S , Q=> , ET=> );
IF (OP30_GVL.OP30_AutoSeq=130 AND OP30_Step_Err_3.Q) THEN
	OP30_GVL.OP30_ErrorWord_0.4:=TRUE;
END_IF

// Checking the gripper condition is opened or not
OP30_Step_Err_3(IN:=OP30_GVL.OP30_AutoSeq=140 , PT:=T#5S , Q=> , ET=> );
IF (OP30_GVL.OP30_AutoSeq=140 AND OP30_Step_Err_3.Q) THEN
	OP30_GVL.OP30_ErrorWord_0.5:=TRUE;
END_IF

//  Horizontal sevo not moving to place position
OP30_Step_Err_3(IN:=OP30_GVL.OP30_AutoSeq=160 , PT:=T#5S , Q=> , ET=> );
IF (OP30_GVL.OP30_AutoSeq=160 AND OP30_Step_Err_3.Q) THEN
	OP30_GVL.OP30_ErrorWord_0.6:=TRUE;
END_IF

//  Vertical sevo not moving to place position
OP30_Step_Err_3(IN:=OP30_GVL.OP30_AutoSeq=180 , PT:=T#5S , Q=> , ET=> );
IF (OP30_GVL.OP30_AutoSeq=180 AND OP30_Step_Err_3.Q) THEN
	OP30_GVL.OP30_ErrorWord_0.7:=TRUE;
END_IF

// Vertical Servo not reaching safe-work position 
OP30_Step_Err_3(IN:=OP30_GVL.OP30_AutoSeq=210 , PT:=T#5S , Q=> , ET=> );
IF (OP30_GVL.OP30_AutoSeq=210 AND OP30_Step_Err_3.Q) THEN
	OP30_GVL.OP30_ErrorWord_0.8:=TRUE;
END_IF

//  Horizontal sevo not moving to safe work position
OP30_Step_Err_3(IN:=OP30_GVL.OP30_AutoSeq=240 , PT:=T#5S , Q=> , ET=> );
IF (OP30_GVL.OP30_AutoSeq=240 AND OP30_Step_Err_3.Q) THEN
	OP30_GVL.OP30_ErrorWord_0.9:=TRUE;
END_IF

END_PROGRAM

// ---- POUs/Programs/OP30/OP30_Initialize_Seq.TcPOU
PROGRAM OP30_Initialize_Seq
VAR
END_VAR

IF OP30_GIUDE_GRP_ctrl.Axis_In_Home AND OP30_GIUDE_GRP_ctrl.Axis_Home_Done AND (SR30_Vert_servo_ctrl.Axis_In_Home) AND OP30_HORI_SERVO_ON_HOME AND NOT OP30_Gripper_LH_State AND NOT OP30_Gripper_RH_State  AND OP30_Gripper_LH_Gripper_ctrl.Axis_reference AND OP30_Gripper_RH_Gripper_ctrl.Axis_reference THEN
	OP30_Temp_hmeOK:=TRUE;
	OP30_HomeRunning:=FALSE;
	OP30_Homing_Seq:=0;
ELSE
	OP30_Temp_hmeOK:=FALSE;	
END_IF

CASE OP30_Homing_Seq OF
	0: IF (OP30_AutoSelected AND NOT OP30_HomeRunning AND NOT OP30_ErrorActive AND NOT OP30_AutoRunning AND NOT OP30_StepRunning AND NOT OP30_Temp_hmeOK) THEN
		OP30_HomeRunning:=TRUE;
		OP30_Homing_Seq:=10;
	   ELSE
		OP30_HomeRunning:=FALSE;	
	   END_IF
	   
	10:IF (OP30_HomeRunning AND (OP30_HMI_Homing OR HMI_Reset))THEN 
		IF (SR30_Vert_servo_ctrl.Axis_In_Home) THEN 
			SR30_Vert_servo_ctrl.Axis_Home_Cmd:=FALSE;
			OP30_Homing_Seq:=20;
		ELSE
			SR30_Vert_servo_ctrl.Position:=0;
			SR30_Vert_servo_ctrl.ABSmove_Start:=TRUE;
	    END_IF	
	   END_IF	
	   
   20: IF (OP30_HORI_SERVO_ON_HOME) THEN 
			SR30_Hori_servo_ctrl.Axis_Home_Cmd:=FALSE;
			OP30_Homing_Seq:=40;
		ELSE
			SR30_HORI_servo_ctrl.Position:=OP30_HORI_SERVO_HME_POS;
			SR30_HORI_servo_ctrl.Velocity:=100;
			SR30_Hori_servo_ctrl.ABSmove_Start:=1;
	    END_IF		
		
   40:  IF  OP30_Gripper_LH_Gripper_ctrl.Axis_reference THEN
		  OP30_Gripper_LH_Close:=1;
		  OP30_Gripper_LH_State:=0;
		  OP30_Homing_Seq:=50;
		ELSE 
			OP30_Gripper_LH_Gripper_ctrl.Reference_Start := TRUE;  
		END_IF
		
   50:	IF  OP30_Gripper_RH_Gripper_ctrl.Axis_reference THEN
			OP30_Gripper_RH_Close:=1;	
   			OP30_Gripper_RH_State:=0;
			OP30_Homing_Seq:=60;
		ELSE
			OP30_Gripper_RH_Gripper_ctrl.Reference_Start := TRUE;	
		END_IF
		
   60: 	CR30_LH_Rej_Cyl.HomingCmd1:=TRUE;	
		IF CR30_LH_Rej_Cyl.Position1 THEN
			CR30_LH_Rej_Cyl.HomingCmd1:=FALSE;
			OP30_Homing_Seq:=70;
		END_IF
		
   70:	CR30_RH_Rej_Cyl.HomingCmd1:=TRUE;	
		IF CR30_RH_Rej_Cyl.Position1 THEN
			CR30_RH_Rej_Cyl.HomingCmd1:=FALSE;
			OP30_Homing_Seq:=75;
		END_IF
		
  75:	IF OP30_GIUDE_GRP_ctrl.Axis_In_Home AND OP30_GIUDE_GRP_ctrl.Axis_Home_Done THEN
	  		OP30_GIUDE_GRP_ctrl.Bsethome:=0;
			OP30_Homing_Seq:=80;
		ELSE
			OP30_GIUDE_GRP_ctrl.Bsethome:=1;
  		END_IF
		
   80:	OP30_Homing_Seq:=0;
   		CR30_LH_Rej_Cyl.HomingCmd1:=FALSE;
   		CR30_RH_Rej_Cyl.HomingCmd1:=FALSE;
		OP30_HomeRunning:=FALSE;
		OP30_HMI_Homing:=FALSE;
END_CASE

END_PROGRAM

// ---- POUs/Programs/OP40/OP40_MAIN.TcPOU
PROGRAM OP40_MAIN
VAR
	OP40_Modeselection_FB: Mode_Selection_Block1;	
//	OP40_Cycle_Time: Cycle_Time_FB;
	TP_100ms: TP;
	Pulse_100ms: BOOL;
	Times: LREAL;
	reset: BOOL;
	Gen_Timer: TON;
END_VAR

// Function Calling

OP40_Manual();
OP40_AUTOSEQUENCE();
OP40_Error();
OP40_Initialization_Seq();
op40_toolchangeover ();
//MOdeselection From HMI

IF (OP40_HMI_AutoMode AND NOT OP40_HMI_ManualMOde AND NOT OP40_HMI_StepMode) THEN
		OP40_Modeselection_FB.ModeWord:=1;
	ELSIF (NOT OP40_HMI_AutoMode AND OP40_HMI_ManualMOde AND NOT OP40_HMI_StepMode) THEN
		OP40_Modeselection_FB.ModeWord:=2;
	ELSIF  (NOT OP40_HMI_AutoMode AND NOT OP40_HMI_ManualMOde AND  OP40_HMI_StepMode) THEN
		OP40_Modeselection_FB.ModeWord:=3;
    ELSE   
		OP40_Modeselection_FB.ModeWord:=0;
END_IF
OP40_Modeselection_FB(
	ModeWord:= , 
	HomeConditionOK:=OP40_HomeConditionOK , 
	OperationEnable:=OP40_AutoSelected, 
	StartPB:=OP40_HMI_Cycle_Start , 
	SafetyAndNOError:= OP40_Safety_OK, 
	ModeAck:=TRUE , 
	HomingINProgress:=OP40_HomeRunning , 
	TempHomeOK:=OP40_Temp_hmeOK , 
	ResetPB:= , 
	AutoSelected=> OP40_AutoSelected, 
	ManualSelected=> OP40_ManualSelected, 
	StepSelected=>OP40_StepSelected , 
	ModeSelAck_Indication=> , 
	StatusDisplay=> , 
	AutoRunning:=OP40_AutoRunning, 
	StepRunning:=OP40_StepRunning , 
	StartEnable:=OP40_StartEnable  , 
	MachineStop:=OP40_Machine_Stop );

OP40_Safety_OK:=OperationEnable;	
	
IF OP40_AutoSelected OR OP40_ManualSelected AND NOT ( OP40_ErrorActive OR OP40_Safety_OK) THEN
	SR40_Vert_servo.bEnable:=TRUE;
ELSE
	SR40_Vert_servo.bEnable:=FALSE;
END_IF

IF OP40_GVL.SR40_Vert_servo.bAxisError OR NOT OP40_Safety_OK  THEN
	OP40_ErrorActive:=TRUE;
END_IF

IF OP40_Stop_Request AND NOT OP40_STN_ENABLE THEN
	OP40_Machine_Stop:=1;
END_IF

Gen_Timer(IN:=OP40_Machine_Stop,PT:=T#5S);
IF Gen_Timer.Q THEN
	OP40_Machine_Stop:=0;
END_IF

END_PROGRAM

// ---- POUs/Programs/OP40/OP40_MANUAL.TcPOU
PROGRAM OP40_MANUAL
VAR
	
    temp_safe:BOOL;
	enable:BOOL;
	reset:bool;
	OP40_Enable: BOOL;
END_VAR


// IF MANUAL IS SELECTED 

//SR40_Vert_servo_ctrl.ABSmove_Start:=OP40_VERT_SERVO_STRT;
OP40_SERVO_POS_DONE			  :=  SR40_Vert_servo_ctrl.pos_done;
OP40_VERT_SERVO_SFE_WRK_POS   :=  OP40_HMI_Safe_Work;
OP40_VERT_SERVO_HME_POS       :=  OP40_HMI_Safe_Home;
OP40_VERT_SERVO_WRK_POS_2     :=  OP40_VERT_SERVO_WORK_POS;
OP40_VERT_SERVO_WRK_POS_1     := (OP40_VERT_SERVO_WORK_POS - OP40_HMI_Servo_Pos_Offset);

IF In_Range(SR40_Vert_servo_status.actualPosition,OP40_VERT_SERVO_SFE_WRK_POS,1) THEN
	OP40_SERVO_ON_SFE_WRK := TRUE;
ELSE
	OP40_SERVO_ON_SFE_WRK := FALSE;
END_IF

IF In_Range(SR40_Vert_servo_status.actualPosition,OP40_VERT_SERVO_HME_POS,1) THEN
	OP40_SERVO_ON_HOME := TRUE;
ELSE
	OP40_SERVO_ON_HOME := FALSE;
END_IF

IF In_Range(SR40_Vert_servo_status.actualPosition,OP40_VERT_SERVO_WRK_POS_1,1) THEN
	OP40_SERVO_ON_WRK_1 := TRUE;
ELSE
	OP40_SERVO_ON_WRK_1 := FALSE;
END_IF

IF In_Range(SR40_Vert_servo_status.actualPosition,OP40_VERT_SERVO_WRK_POS_2,1) THEN
	OP40_SERVO_ON_WRK_2 := TRUE;
ELSE
	OP40_SERVO_ON_WRK_2 := FALSE;
END_IF

SR40_Vert_servo(
	bAxis1_Ref_Switch:= , 
	bInit:= , 
	bErrorReset:= OP40_HMI_Reset OR Servo_Reset , 
	bEnable:=Servo_Enable , 
	bMoveVelocity:= , 
	bHalt:=  , 
	bManualMode:= MANUAL_SELECTED AND OP40_ManualSelected, 
	fHomePos:= , 
	fOverride:= , 
	fTargetPosition:= SR40_Vert_servo_ctrl.Position, 
	fTargetVelocity:= SR40_Vert_servo_ctrl.Velocity, 
	fAcc:= , 
	fDec:= , 
	Servo_High_Limit:= OP40_HMI_High_Limit,	
	Servo_Low_Limit:=  OP40_HMI_Low_Limit,
	WARNING_LIMIT:=1,	
	Safe_move_Conditions:= Servo_Safety, 
	Axis:= SR40_Vert_servo_Axis, 
	HME_WRITE_ADD:= 16#5004,
	bHome:= SR40_Vert_servo_ctrl.Bsethome , 
	bSetPosition:= SR40_Vert_servo_ctrl.Bsetpos  , 
	bMoveAbsolute:= SR40_Vert_servo_ctrl.ABSmove_Start, 
	bMoveRelative:= SR40_Vert_servo_ctrl.RELmove_Start, 
	bMoveTorque:= SR40_Vert_servo_ctrl.Torque_mode_Start, 
	stManualModeAxis:= SR40_Vert_servo_status , 
	bmove_home:= SR40_Vert_servo_ctrl.Axis_Home_Cmd , 
	sAxisState=> SR40_Vert_servo_ctrl.Axis_State , 
	bAxis_ready=> SR40_Vert_servo_ctrl.Axis_ready , 
	bAxisInPosition=> SR40_Vert_servo_ctrl.Axis_In_Pos , 
	bAxisError=> SR40_Vert_servo_ctrl.Axis_Error , 
	bAxisEnabled=> SR40_Vert_servo_ctrl.Axis_Enabled, 
	bAxisHomed=> SR40_Vert_servo_ctrl.Axis_reference , 
	bSetPositionDone=> , 
	bHaltDone=>  SR40_Vert_servo_ctrl.Axis_Halted , 
	bSTOPDone=> , 
	bHomeDone=> , 
	bDone=> , 
	bTorqueReached=> , 
	bsafe_to_move=> , 
	baxis_in_home_pos=> SR40_Vert_servo_ctrl.Axis_In_Home , 
	bABS_Pos_done=>SR40_Vert_servo_ctrl.pos_done , 
	Actual_position=>SR40_Vert_servo_ctrl.Actual_Position ,  
	Actual_velocity=>SR40_Vert_servo_ctrl.Actual_Velocity , 
	Actual_Torque=> SR40_Vert_servo_ctrl.Actual_Torque);
	
IF MANUAL_SELECTED AND OP40_ManualSelected THEN	
	SR40_Vert_servo_status.targetVelocity:=50;	
END_IF

OP40_LH_LVDT_VALUE := DINT_TO_REAL(OP40_LH)/10000;
OP40_RH_LVDT_VALUE := DINT_TO_REAL(OP40_RH)/10000;

END_PROGRAM

// ---- POUs/Programs/OP40/OP40_AUTOSEQUENCE.TcPOU
PROGRAM OP40_AUTOSEQUENCE
VAR

//INT

	OP40_FIXTURE_2					: INT;
	OP40_FIXTURE_1					: INT;
	Dry_run: BOOL;	
	
// TIMER
	OP40_AFT_WRK_POS : TON;

	OP40_STN_MOVER: INT;
	MOVER_POS_RECHED_R: R_TRIG;
	
	OP40_Cycle_Time_FB : FB_Cycletime;	
END_VAR


IF (NOT OP40_AutoSelected) OR (OP40_ErrorActive OR OP40_HomeRunning ) OR NOT OperationEnable THEN
	OP40_AutoRunning:= FALSE;
	OP40_AutoSeq:= 10;
//	OP40_STN_ENABLE:=FALSE;
END_IF	


CASE OP40_AutoSeq OF
		
		10: IF (OP40_AutoSelected) THEN		// Check Automode Selected
				OP40_AutoSeq:=20;
	        END_IF
		
	    20:IF ( NOT OP40_ErrorActive) THEN		//Check No error
		       OP40_AutoSeq:=30;
      	   END_IF
		   
      	30:IF (NOT OP40_HomeRunning) THEN		//Check No Homerunning
      		   OP40_AutoSeq :=40;
      	   END_IF
		   
        40:IF (OP40_Main.OP40_Modeselection_FB.TempHomeOK)THEN	//Check Machine in Home
      		   OP40_AutoSeq:= 50;
      	   END_IF
		   
      	50:IF ( OP40_STN_ENABLE AND OP40_STN_RUNNING ) THEN		// Check Operation Completed Reset
      		   OP40_AutoSeq:=70;
		   ELSE
	   		   OP40_AutoSeq:=60;
      	   END_IF
		   
	   60:IF (AUTO_RUNNING OR (NOT AUTO_RUNNING AND OP40_HMI_Cycle_Start)) THEN		//Machine Start in Fully Automatic or Press Cycle Start For Semi Automatic
		    OP40_HomeConditionOK:=TRUE;
	 			IF( OP40_Main.OP40_Modeselection_FB.HomeConditionOK AND OP40_AutoSelected) THEN
					OP40_AutoRunning:=TRUE;
					OP40_StepRunning:= FALSE;		
				ELSIF (OP40_Main.OP40_Modeselection_FB.HomeConditionOK AND OP40_StepSelected) THEN
					OP40_AutoRunning:=FALSE;
					OP40_StepRunning:= TRUE;
				END_IF;
		  END_IF
		  
		  IF ((OP40_AutoRunning OR OP40_StepRunning) AND OP40_StartEnable) THEN
			OP40_AutoSeq:= 70;
		  END_IF	

      	70:  // SERVO POSITION SAFE CHECK
	       IF (OP40_SERVO_ON_SFE_WRK OR OP40_SERVO_ON_HOME) AND NOT SR40_Vert_servo_ctrl.ABSmove_Start THEN 
	        SR40_Vert_servo_ctrl.Position:=OP40_VERT_SERVO_WRK_POS_1;   
	        OP40_AutoSeq:=75;
	       END_IF
		   
		75: // WAITING FOR MOVER AND MOVING SERVO TO TARGET POSITION
			IF OP40_STN_ENABLE AND SR40_Vert_servo_ctrl.Position=OP40_VERT_SERVO_WRK_POS_1 THEN
			 SR40_Vert_servo_ctrl.Velocity:=OP40_HMI_Servo_Speed;
			 OP40_STN_RUNNING:=1;
			 SR40_Vert_servo_ctrl.ABSmove_Start:=TRUE;
			 IF OP40_FIXTURE_1=30 OR OP40_FIXTURE_2=30 THEN
			 	OP40_AutoSeq:=80;
			 ELSIF OP40_FIXTURE_1<>30 AND OP40_FIXTURE_2<>30 THEN
				OP40_AutoSeq:=76;
			 END_IF
			END_IF
			
		76: OP40_STN_ENABLE:=0;
			IF 	(MOVER_CMP_STATUS[OP40_STN_MOVER][1]=41 AND MOVER_CMP_STATUS[OP40_STN_MOVER][2]=41) THEN
				MOVER_STP_NO[OP40_CURR_MOVER]	:= (OP160_XTS_POS_NO*10);
			ELSE		
				STATION_DONE[OP40_CURR_MOVER][OP40_XTS_POS_NO]	:= TRUE;
			END_IF	
			IF MOVER_STP_NO[OP40_CURR_MOVER]<>((OP40_XTS_POS_NO*10)+1)THEN 
				OP40_CURR_MOVER	:= 0;
				OP40_AutoSeq	:= 75;  
			END_IF		
			
		80:  IF SR40_Vert_servo_ctrl.pos_done AND OP40_SERVO_ON_WRK_1 THEN
			   SR40_Vert_servo_ctrl.ABSmove_Start:=FALSE;
			   SR40_Vert_servo_ctrl.Position:=OP40_GVL.OP40_VERT_SERVO_WRK_POS_2;
			   SR40_Vert_servo_ctrl.Velocity:=(OP40_HMI_Servo_Speed-OP40_HMI_Servo_Speed_Offset);
			   OP40_AutoSeq:=90;
			 ELSIF SR40_Vert_servo_ctrl.pos_done AND OP40_SERVO_ON_WRK_2 THEN
 				OP40_AutoSeq:=100;
			 END_IF
			  
		90: IF OP40_SERVO_ON_WRK_1 AND NOT SR40_Vert_servo_ctrl.ABSmove_Start THEN                   
               SR40_Vert_servo_ctrl.ABSmove_Start:=TRUE; 
			    OP40_LH_LVDT_OK:=0;
				OP40_LH_LVDT_NOK:=0;
				OP40_RH_LVDT_OK:=0;
				OP40_RH_LVDT_NOK:=0;
               OP40_AutoSeq:=100;
			END_IF
			
		100: // START THE SPINNER OK COMPONENT FIXTURE
			IF OP40_AFT_WRK_POS.Q AND OP40_SERVO_ON_WRK_2 THEN	
			 SR40_Vert_servo_ctrl.ABSmove_Start:=FALSE;		 
			  IF OP40_FIXTURE_1=30 THEN
			 	 IF In_Range(OP40_LH_LVDT_VALUE,OP40_SET_LVDT_VALUE,OP40_LVDT_TOLERANCE) THEN
				  OP40_LH_LVDT_OK  := 1;
				  OP40_LH_LVDT_NOK := 0;				  				  
			 	 ELSE
				  OP40_LH_LVDT_NOK := 1;
				  OP40_LH_LVDT_OK  := 0;
			 	 END_IF  
			  END_IF
			  IF OP40_FIXTURE_2=30 THEN
			  	IF In_Range(OP40_RH_LVDT_VALUE,OP40_SET_LVDT_VALUE,OP40_LVDT_TOLERANCE) THEN
				  OP40_RH_LVDT_OK  := 1;
				  OP40_RH_LVDT_NOK := 0;			  				  
			  	ELSE
				  OP40_RH_LVDT_NOK := 1;
				  OP40_RH_LVDT_OK  := 0;
			    END_IF
		 	  END_IF
				OP40_HMI_LH_LVDT_VALUE:=OP40_LH_LVDT_VALUE;
				OP40_HMI_RH_LVDT_VALUE:=OP40_RH_LVDT_VALUE;			  
			  IF NOT SR40_Vert_servo_ctrl.ABSmove_Start THEN
				 SR40_Vert_servo_ctrl.Position:=OP40_VERT_SERVO_SFE_WRK_POS;
				 SR40_Vert_servo_ctrl.Velocity:=OP40_HMI_Servo_Speed;
				 OP40_AutoSeq:=110;
			  END_IF				    			  
		    END_IF
			OP40_CURR_MOVER				:= OP40_STN_MOVER;
		
		110: // SERVO MOVE TO SAFE WORK POSITION	 
			IF NOT SR40_Vert_servo_ctrl.ABSmove_Start AND SR40_Vert_servo.fTargetPosition=OP40_VERT_SERVO_SFE_WRK_POS THEN
				SR40_Vert_servo_ctrl.ABSmove_Start:=TRUE;
			 IF OP40_FIXTURE_1=30 THEN
				IF OP40_LH_LVDT_OK THEN
					MOVER_CMP_STATUS[OP40_CURR_MOVER][1]:=40;
				ELSIF OP40_LH_LVDT_NOK THEN  
					MOVER_CMP_STATUS[OP40_CURR_MOVER][1]:=41;	
				END_IF
			 END_IF	
			 IF OP40_FIXTURE_2=30 THEN
				IF OP40_RH_LVDT_OK THEN
					MOVER_CMP_STATUS[OP40_CURR_MOVER][2]:=40;
				ELSIF OP40_RH_LVDT_NOK THEN  
					MOVER_CMP_STATUS[OP40_CURR_MOVER][2]:=41;	
				END_IF	
			END_IF		
				OP40_STN_ENABLE:=FALSE;	
				OP40_AutoSeq:=120;
			END_IF
				
		120: // SERVO DONE
			IF SR40_Vert_servo_ctrl.pos_done AND OP40_SERVO_ON_SFE_WRK THEN
			 	SR40_Vert_servo_ctrl.ABSmove_Start:=FALSE;
				OP40_STN_RUNNING:=0;
			 	OP40_STN_ENABLE:=FALSE;
			IF 	(MOVER_CMP_STATUS[OP40_STN_MOVER][1]=41 AND MOVER_CMP_STATUS[OP40_STN_MOVER][2]=41) THEN
				MOVER_STP_NO[OP40_CURR_MOVER]	:= (OP160_XTS_POS_NO*10);
			ELSE
				STATION_DONE[OP40_CURR_MOVER][OP40_XTS_POS_NO]	:= TRUE;				
			END_IF	
			END_IF	
			IF MOVER_STP_NO[OP40_CURR_MOVER]<>((OP40_XTS_POS_NO*10)+1)THEN
			OP40_CURR_MOVER		:= 0;
			 OP40_AutoSeq		:=70;
			END_IF
END_CASE 


OP40_Cycle_Time_FB(i_b_startTime:=OP40_STN_ENABLE , i_b_stopTime:= NOT OP40_STN_ENABLE , o_t_StationTime=>OP40_Cycle_time );					

Dry_Run:=All_Station_Dry_Run;
IF Dry_run THEN
	OP40_FIXTURE_1:=30;
    OP40_FIXTURE_2:=30;
ELSE
	OP40_FIXTURE_1:=MOVER_CMP_STATUS[OP40_STN_MOVER][1];
	OP40_FIXTURE_2:=MOVER_CMP_STATUS[OP40_STN_MOVER][2];	
END_IF




OP40_AFT_WRK_POS(IN:=(OP40_SERVO_ON_WRK_2 AND (OP40_AutoSeq=100)), PT:=INT_TO_TIME(OP40_DLY_AFT_SFE_WRK) , Q=> , ET=> );
//Timer(IN:=OP40_STN_ENABLE,PT:=T#10S);



////################################ STATION ENABLE CONTION    ############################
	OP40_STN_MOVER					:= MOVER_POSITION[OP40_XTS_POS_NO];
IF AUTO_WITH_XTS THEN		
IF OP40_STN_MOVER>0 THEN
IF NOT(END_OF_CYCLE AND MOVER_CMP_STATUS[OP40_STN_MOVER][1]=5 AND MOVER_CMP_STATUS[OP40_STN_MOVER][2]=5)THEN	 
	OP40_STN_ENABLE					:= MOVER_POS_RECHED[OP40_STN_MOVER] AND ((MOVER_CMP_STATUS[OP40_STN_MOVER][1]=30)OR 
										(MOVER_CMP_STATUS[OP40_STN_MOVER][2]=30)) AND STATION_ENABLE_CONTROL;
ELSE
	STATION_DONE[OP40_STN_MOVER][OP40_XTS_POS_NO]			:= TRUE;
END_IF
ELSE
	OP40_STN_ENABLE					:= FALSE;
END_IF																			
END_IF

END_PROGRAM

// ---- POUs/Programs/OP40/OP40_ERROR.TcPOU
PROGRAM OP40_ERROR
VAR
	OP40_StepErr_1: TON;
	OP40_Step_Err_2: TON;
	OP20_StepErr_3 : TON;
END_VAR


// Set ERROR ACTIVE
IF ((OP40_GVL.OP40_ErrorWord_0<>0) OR (OP40_GVL.OP40_ErrorWord_1<>0) OR (OP40_GVL.OP40_ErrorWord_2<>0)) THEN
	OP40_GVL.OP40_ErrorActive:= TRUE;
	END_IF

//Reset ErrorActive
IF (OP40_HMI_Reset OR HMI_Reset) THEN 
	OP40_GVL.OP40_ErrorActive:= FALSE;
	OP40_GVL.OP40_ErrorWord_0:= 0;
	OP40_GVL.OP40_ErrorWord_1:= 0;
	OP40_GVL.OP40_ErrorWord_2:= 0;

END_IF

OP40_ErrorWord_0.0:=SR40_Vert_servo.bAxisError;
OP40_ErrorWord_0.1:=NOT OperationEnable;

// Auto Seq Step Error
//Servo not reaching work position
//OP40_StepErr_1(IN:=(OP40_AutoSeq=80) , PT:=T#1S , Q=> , ET=> );
//IF (OP40_AutoSeq=80 AND NOT OP40_GVL.OP40_SERVO_ON_WRK_1 AND OP40_StepErr_1.Q) THEN
//	OP40_GVL.OP40_ErrorWord_0.2:=TRUE;
//END_IF

// Servo Not Reached home position or safe-work position
OP40_Step_Err_2(IN:=OP40_AutoSeq=120 , PT:=T#5S , Q=> , ET=> );
IF (OP40_AutoSeq=120 AND NOT SR40_Vert_servo_ctrl.Axis_In_Home AND OP40_Step_Err_2.Q) THEN
	OP40_GVL.OP40_ErrorWord_0.3:=TRUE;
END_IF

//OP20_StepErr_3(IN:=( OP40_HomeRunning AND (OP40_Homing_Seq=10)), PT:=T#5S , Q=> , ET=> );
//IF OP20_StepErr_3.Q THEN
//	OP20_GVL.OP20_ErrorWord_0.4:=TRUE;
//END_IF

END_PROGRAM

// ---- POUs/Programs/OP40/OP40_Initialization_Seq.TcPOU
PROGRAM OP40_Initialization_Seq
VAR
END_VAR

IF (SR40_Vert_servo_ctrl.Axis_In_Home)THEN
    OP40_Temp_hmeOK:=TRUE;
	OP40_HomeRunning:=FALSE;
	OP40_Homing_Seq:=0;
ELSE
	OP40_Temp_hmeOK:=FALSE;	
END_IF

CASE OP40_Homing_Seq OF
	0: IF (OP40_AutoSelected AND NOT OP40_HomeRunning AND NOT OP40_ErrorActive AND NOT  OP40_AutoRunning AND NOT OP40_StepRunning AND NOT OP40_Temp_hmeOK ) THEN
		OP40_HomeRunning:=TRUE;
		OP40_Homing_Seq:=10;	
	   END_IF
	10:IF (OP40_HomeRunning AND (OP40_HMI_Homing OR HMI_Reset))THEN 
		IF (SR40_Vert_servo_ctrl.Axis_In_Home) THEN 
			OP40_Homing_Seq:=20;
			SR40_Vert_servo_ctrl.Axis_Home_Cmd:=FALSE;
		ELSE
			SR40_Vert_servo_ctrl.Position:=0;
			SR40_Vert_servo_ctrl.Velocity:=100;
			SR40_Vert_servo_ctrl.ABSmove_Start:=TRUE;
			SR40_Vert_servo_ctrl.Axis_Home_Cmd:=TRUE;
	    END_IF
	   END_IF		
	20:	OP40_Homing_Seq:=0;
		OP40_HomeRunning:=FALSE;
	
END_CASE

END_PROGRAM

// ---- POUs/Programs/OP40/op40_toolchangeover.TcPOU
PROGRAM op40_toolchangeover
VAR
	op40_tool_change                    : tool_changeover;
	OP40_TOOL_CHANGE_MODE_SELECTED      : bool;
	fb_reset_1                          : BOOL;
	tool_6_fb                           : BOOL;
	tool_8_fb                           : BOOL;
	OP40_TOL_UNLOD_STRT					: BOOL;
	OP40_TOL_LOAD_STRT					: BOOL;
	OP40_TOL_DISENGAGE					: BOOL;
	OP40_TOL_ENGAGE						: BOOL;
	op40_manual_lock                    : BOOL;
	op40_manual_unlock                  : BOOL;
	OP40_UNLD_STUS                      : STRING;
	OP40_LOAD_STUS                      : STRING;
END_VAR

VAR PERSISTENT
	
	OP40_TOL_WRK_POS					: LREAL;
	OP40_TOL_HME_POS					: LREAL;
	op40_TOL_VELOCITY					: LREAL;
	OP40_TOL_CHNGE_CMPLE				: BOOL;
	OP40_TOL_LOAD_COMPLE                : BOOL;
	OP40_TOL_UNLOAD_COMPLE              : BOOL;
	
END_VAR

IF OP40_TOOL_CHANGE_MODE_SELECTED THEN

op40_tool_change(
	actual_pos:=SR40_Vert_servo_ctrl.Actual_Position,
	actual_vel:=SR40_Vert_servo_ctrl.Actual_Velocity,
	target_work_pos:= OP40_TOL_WRK_POS, 
	target_home_pos:= OP40_TOL_HME_POS, 
	target_vel_from_hmi:= op40_TOL_VELOCITY, 
	station_number:= , 
	mover_number:= , 
	no_of_mover_present:= , 
	model_selected:= model_selected, 
	tool_unloading_start:=OP40_TOL_UNLOD_STRT , 
	tool_loading_start:=OP40_TOL_LOAD_STRT , 
	error_active:= , 
	station_in_auto:= OP40_AutoSelected, 
	station_in_home:=  , 
	absoulte_move_done:= SR40_Vert_servo_ctrl.Axis_In_Pos, 
	tool_6_3_present:= tool_6_fb, 
	tool_7_89_present:= tool_8_fb, 
	fb_reset:=fb_reset_1,
	SERVO_TOL_CHECK_OFFSET_POS := 18, 
	tool_changer_over_complete=> OP40_TOL_CHNGE_CMPLE,
	tool_disengage=> OP40_TOL_DISENGAGE, 
	tool_engagae=> OP40_TOL_ENGAGE, 
	tool_loading_complete=> OP40_TOL_LOAD_COMPLE, 
	tool_unloading_complete=> OP40_TOL_UNLOAD_COMPLE, 
	servo_move_abs=>SR40_Vert_servo_ctrl.ABSmove_Start, 
	unloading_status=>OP40_UNLD_STUS , 
	loading_status=>OP40_LOAD_STUS , 
	target_pos_to_servo=> SR40_Vert_servo_ctrl.Position, 
	target_vel_to_servo=> SR40_Vert_servo_ctrl.Velocity,
    tool_loading_failed := );
	
END_IF	

IF op40_manual_lock OR OP40_TOL_ENGAGE THEN
	O40_TOOL_CHO_UNLOCK_Q1151_0     :=0;
	O40_TOOL_CHO_LOCK_Q1151_1       :=1;
ELSIF op40_manual_unlock OR OP40_TOL_DISENGAGE THEN
	 O40_TOOL_CHO_UNLOCK_Q1151_0     :=1;
	 O40_TOOL_CHO_LOCK_Q1151_1       :=0;
END_IF

END_PROGRAM

// ---- FB/tool/tool_changeover.TcPOU
FUNCTION_BLOCK tool_changeover
VAR_INPUT 
	// LREAL
	actual_pos                 : LREAL;
	actual_vel                 : LREAL;
	target_work_pos            : LREAL;
	target_home_pos            : LREAL;
	target_vel_from_hmi        : LREAL;
	SERVO_TOL_CHECK_OFFSET_POS : LREAL;	
	//INT
	station_number             : INT;
	mover_number               : INT;
	no_of_mover_present        : INT;
	model_selected             : INT;
	
	//BOOL
	tool_unloading_start       : BOOL;
	tool_loading_start         : BOOL;
	error_active               : BOOL;
	station_in_auto            : BOOL;
	station_in_home            : BOOL;
	absoulte_move_done         : BOOL;
	tool_6_3_present           : BOOL;
	tool_7_89_present          : BOOL;
	fb_reset                   : BOOL;
    operator_ack               : BOOL;
	
END_VAR                        

VAR_OUTPUT PERSISTENT
	tool_changer_over_complete : BOOL;
	tool_disengage             : BOOL;
	tool_engagae               : BOOL;
	tool_loading_complete		: BOOL;
	tool_unloading_complete    : BOOL;
	servo_move_abs             : BOOL;
	tool_loading_failed        : BOOL;
	unloading_status           : STRING;
	loading_status             : STRING;
	
	target_pos_to_servo        : LREAL;
	target_vel_to_servo        : LREAL;
	
END_VAR

VAR PERSISTENT
	//INT
	Unloading_Sequence         : INT;
	Loading_Sequence           : INT;
	model_present              : INT;
	
	// BOOL
	target_pos_reached		   : BOOL;
	engaged_check              : BOOL;
	unloading_started          : BOOL; 
	loading_started            : BOOL;
	disengage_check            : BOOL;
	//TIMER
	disengage_timer            :ton;
	engage_timer               :ton;
	disengae_timer             :TON;
	
	
END_VAR

VAR
	SERVO_WRK_POS				: BOOL;
	SERVO_HME_POS				: BOOL;
	SERVO_TOL_CHCK_POS          : BOOL;
	dis: BOOL;
END_VAR
VAR_IN_OUT
	
END_VAR

                                    ////////////////////////////////////// GENERAL SEQUENCE //////////////////////////////////////

IF (error_active AND station_in_auto) THEN
	tool_disengage             := FALSE;
	tool_engagae               := FALSE;
	servo_move_abs             := FALSE;
	unloading_status           := 'error active clear error';
	
ELSIF  NOT error_active AND NOT station_in_auto THEN
		unloading_status       := 'station is not in auto';
		
ELSIF NOT error_active AND station_in_auto AND station_in_home AND NOT unloading_started AND NOT loading_started THEN
	  Unloading_Sequence        := 0;
	  loading_Sequence          := 0;
	  
	  IF tool_changer_over_complete THEN
	  tool_changer_over_complete := FALSE;
	  END_IF
END_IF

                         ////////////////////////////////////////// block complete reset //////////////////////////////////////////
						 
IF fb_reset THEN
	tool_changer_over_complete := FALSE;
	tool_disengage             := false;
	tool_engagae               := false;
	tool_loading_complete      := false;
	tool_unloading_complete    := false;
	servo_move_abs             := FALSE;
	SERVO_WRK_POS			   := FALSE;
	SERVO_HME_POS			   := FALSE;
	SERVO_TOL_CHCK_POS         := FALSE;
	engaged_check              := FALSE;
	unloading_started          := FALSE;	
	unloading_status           := 'block reseted';
	loading_status             := 'block reseted';
	target_pos_to_servo        := 0.0;
	target_vel_to_servo		   := 0.0;
    Unloading_Sequence         := 0;
    loading_Sequence           := 0;	
END_IF 

               ////////////////////////////////////////////////////// model selected ///////////////////////////////////////////////////////////
			   
// model number = 1 then tool for 6.3 present
// model number = 2 then tool for 7.89 present	
	   
IF tool_6_3_present AND NOT tool_7_89_present THEN
	  model_present :=1;
ELSIF tool_7_89_present AND NOT tool_6_3_present THEN
	  model_present :=2;
END_IF


                            ////////////////////////////////////// UNLOADING SEQUENCE //////////////////////////////////////////
							
CASE Unloading_Sequence OF
	
     0: IF NOT tool_loading_complete  AND NOT tool_unloading_complete  AND	tool_unloading_start THEN          // check tool change over start command
		       unloading_started := TRUE;
               Unloading_Sequence := 10;
	    ELSIF NOT tool_unloading_start THEN
	          unloading_status := 'waiting for tool unloading start command';
		ELSIF NOT tool_unloading_complete THEN
			 unloading_status := 'previous unloading complete bit is not reseted';
		ELSIF NOT tool_loading_complete THEN
			 unloading_status := 'previous loading complete bit is not reseted';	 
	 END_IF
	 
	 
	 10: IF model_selected = model_present THEN
		   Unloading_Sequence  :=  60;
		ELSIF model_selected <> model_present THEN
			Unloading_Sequence  :=  20;
	    END_IF
	 
     20: target_pos_to_servo := target_work_pos ;                                                              // moving target position and velocity to servo 
         target_vel_to_servo := target_vel_from_hmi ;
		 
		 IF target_pos_to_servo = target_work_pos AND target_vel_to_servo = target_vel_from_hmi THEN
			 servo_move_abs      := TRUE;
			 unloading_status    := ' target position and velocity to servo moved ';
			 Unloading_Sequence  :=  30;
	     ELSIF target_pos_to_servo <> target_work_pos OR target_vel_to_servo <> target_vel_from_hmi THEN	
		      unloading_status   := ' target position or velocity to servo not moved ';
		 END_IF
		 
	 30: IF  absoulte_move_done AND SERVO_WRK_POS  THEN
		 
		     servo_move_abs := FALSE;
             tool_disengage := TRUE;
			 Unloading_Sequence  := 40;
			 
		 ELSIF NOT absoulte_move_done AND SERVO_WRK_POS THEN 
			   unloading_status   := ' waiting for absolute done ';
	     ELSIF 	absoulte_move_done AND NOT SERVO_WRK_POS THEN 
			 unloading_status   := ' waiting target pos reached fb ';		 
		 END_IF 	 
		
	 40: IF disengage_timer.Q THEN
		    target_pos_to_servo := target_work_pos - SERVO_TOL_CHECK_OFFSET_POS;                                                              
            target_vel_to_servo := target_vel_from_hmi ;
			
             IF target_pos_to_servo = target_work_pos- SERVO_TOL_CHECK_OFFSET_POS AND target_vel_to_servo = target_vel_from_hmi THEN
			  servo_move_abs      := TRUE;
			  Unloading_Sequence  := 50;
			  unloading_status    := ' target position and velocity to servo moved ';
			  
			  ELSIF target_pos_to_servo <> target_work_pos- SERVO_TOL_CHECK_OFFSET_POS OR target_vel_to_servo <> target_vel_from_hmi THEN
				     unloading_status   := ' target position or velocity to servo not moved ';
		     END_IF
			
		ELSIF NOT disengage_timer.Q THEN
			  unloading_status   := ' waiting for 5s  ';
	    END_IF
		
		
     50: IF absoulte_move_done  AND SERVO_TOL_CHCK_POS THEN
		    servo_move_abs := FALSE;
		    Unloading_Sequence  := 60;
			
		ELSIF NOT absoulte_move_done AND SERVO_TOL_CHCK_POS THEN 
			   unloading_status   := ' waiting for absolute done ';
			   
	     ELSIF 	absoulte_move_done AND NOT SERVO_TOL_CHCK_POS THEN 
			 unloading_status   := ' waiting target pos reached fb ';	
	 END_IF

  
	 60: IF  model_present = 1  THEN
		     IF NOT tool_6_3_present THEN
                    tool_disengage := FALSE;
			        target_pos_to_servo := target_home_pos;                                                              
                    target_vel_to_servo := target_vel_from_hmi;
			        unloading_status   := ' tool disengaged ';	
			     IF target_pos_to_servo = target_home_pos AND target_vel_to_servo = target_vel_from_hmi THEN
			      servo_move_abs      := TRUE;
			      Unloading_Sequence  := 70;  
			     ELSIF target_pos_to_servo <> target_home_pos OR target_vel_to_servo <> target_vel_from_hmi THEN
	                 unloading_status   := ' target position or velocity to servo not moved ';
		         END_IF	  
 
			 ELSIF  tool_6_3_present THEN
				    unloading_status   := ' tool not disengaged ';
			 END_IF 
			 
		 ELSIF  model_present = 2 THEN
			   IF NOT  tool_7_89_present THEN
				       tool_disengage := FALSE;
			           target_pos_to_servo := target_home_pos;                                                              
                       target_vel_to_servo := target_vel_from_hmi;
			           unloading_status   := ' tool disengaged ';  
			       IF target_pos_to_servo = target_home_pos AND target_vel_to_servo = target_vel_from_hmi THEN
			          servo_move_abs      := TRUE;
			          Unloading_Sequence  := 70;
			        ELSIF target_pos_to_servo <> target_home_pos OR target_vel_to_servo <> target_vel_from_hmi THEN
	                  unloading_status   := ' target position or velocity to servo not moved ';
		           END_IF
			   
			   ELSIF  tool_7_89_present THEN
				       unloading_status   := ' tool not disengaged ';
			   
			   END_IF
	 
		 END_IF

		
     70: IF  absoulte_move_done AND SERVO_HME_POS  THEN
     		 
     		     servo_move_abs         := FALSE;
     	         Unloading_Sequence     := 80;
				 
         ELSIF NOT absoulte_move_done AND SERVO_HME_POS THEN 
     			   unloading_status   := ' waiting for absolute done ';
     			   
     	 ELSIF 	absoulte_move_done AND NOT SERVO_HME_POS THEN 
     			 unloading_status   := ' waiting target pos reached fb ';
     		 
     	 END_IF

     80: IF  NOT tool_7_89_present AND NOT tool_6_3_present THEN
             tool_unloading_complete:= TRUE;
             model_present :=0;
		 END_IF
		 
END_CASE


                               ////////////////////////////////////// LOADING SEQUENCE /////////////////////////////////////////////
							   
CASE loading_sequence OF
	
	0: IF 	tool_loading_start AND tool_unloading_complete AND model_present = 0 AND Unloading_Sequence = 80 THEN
		    loading_Sequence := 10;
	    ELSIF NOT 	tool_loading_start AND tool_unloading_complete AND model_present = 0 THEN
	          loading_status := 'waiting for tool chageover start command';
	    ELSIF tool_loading_start AND NOT tool_unloading_complete AND model_present = 0 THEN
		       loading_status := 'waiting for tool unloding complete feedback';
		ELSIF tool_loading_start AND  tool_unloading_complete AND  model_present <> 0	THEN
              loading_status := 'model present is not equal to 0 ';
	 END_IF
	 
     10: target_pos_to_servo := target_work_pos ;                                                              // moving work position and velocity to servo 
         target_vel_to_servo := target_vel_from_hmi ;
		 tool_disengage      := TRUE ;
		 
		 IF target_pos_to_servo = target_work_pos AND target_vel_to_servo = target_vel_from_hmi THEN
			 servo_move_abs      := TRUE;
			 loading_status    := ' target position and velocity to servo moved ';
			 loading_Sequence  :=  20;
	     ELSIF target_pos_to_servo <> target_work_pos OR target_vel_to_servo <> target_vel_from_hmi THEN	
		      loading_status   := ' target position or velocity to servo not moved ';
		 END_IF
		 
	 20: IF  absoulte_move_done AND SERVO_WRK_POS  THEN
		 
		     servo_move_abs := FALSE;
			 engaged_check  := TRUE ;
			 tool_disengage := FALSE ;
			 tool_engagae   := TRUE;
			 loading_Sequence  := 30;
			 
		 ELSIF NOT absoulte_move_done AND SERVO_WRK_POS THEN 
			   loading_status   := ' waiting for absolute done ';
	     ELSIF 	absoulte_move_done AND NOT SERVO_WRK_POS THEN 
			 loading_status   := ' waiting target pos reached fb ';		 
		 END_IF 	 
		
	 30: IF engage_timer.q THEN
		    target_pos_to_servo := target_work_pos - SERVO_TOL_CHECK_OFFSET_POS;          // moving enage position and velocity to servo                                                     
            target_vel_to_servo := target_vel_from_hmi ;
			engaged_check       := FALSE;
             IF target_pos_to_servo = target_work_pos- SERVO_TOL_CHECK_OFFSET_POS AND target_vel_to_servo = target_vel_from_hmi THEN
			  servo_move_abs      := TRUE;
			  loading_Sequence  := 40;
			 ELSIF target_pos_to_servo <> target_work_pos- SERVO_TOL_CHECK_OFFSET_POS OR target_vel_to_servo <> target_vel_from_hmi THEN 
				   loading_status   := ' target position or velocity to servo not moved ';
		     END_IF
			
	    END_IF
		
		
	 
	 40: IF  absoulte_move_done AND SERVO_TOL_CHCK_POS  THEN
		     servo_move_abs := FALSE;
			 loading_Sequence  := 50;
		 ELSIF NOT absoulte_move_done AND SERVO_TOL_CHCK_POS THEN 
			   loading_status   := ' waiting for absolute done ';   
	     ELSIF 	absoulte_move_done AND NOT SERVO_TOL_CHCK_POS THEN 
			 loading_status   := ' waiting target pos reached fb ';	
		 END_IF

	         
	 
		 50: IF model_selected=1 THEN                       // moving home position and velocity to servo  
                   IF tool_6_3_present AND  model_present = 1 THEN
				   target_pos_to_servo := target_home_pos;                                                              
                   target_vel_to_servo := target_vel_from_hmi;
			 
			        IF target_pos_to_servo = target_home_pos AND target_vel_to_servo = target_vel_from_hmi THEN
			           servo_move_abs      := TRUE;
			           loading_Sequence  := 60;
					   
					ELSIF target_pos_to_servo <>  target_home_pos AND target_vel_to_servo <> target_vel_from_hmi THEN  
                            loading_status   := ' target position or velocity to servo not moved '; 
		             END_IF
				   ELSIF NOT (tool_6_3_present AND tool_7_89_present) OR  model_present <> 1 THEN
	                     loading_status   :='tool not engaged';
					ELSIF (NOT tool_6_3_present AND tool_7_89_present) AND  model_present <> 1 THEN
						   loading_Sequence  := 101;
				END_IF
				
             ELSIF model_selected=2 THEN
				   IF tool_7_89_present AND  model_present = 2 THEN
					  target_pos_to_servo := target_home_pos;                                                              
                      target_vel_to_servo := target_vel_from_hmi;
			 
			          IF target_pos_to_servo = target_home_pos AND target_vel_to_servo = target_vel_from_hmi THEN
			           servo_move_abs      := TRUE;
			           loading_Sequence  := 60;
					  ELSIF target_pos_to_servo <>  target_home_pos AND target_vel_to_servo <> target_vel_from_hmi THEN  
                            loading_status   := ' target position or velocity to servo not moved '; 
		             END_IF
					 
					 ELSIF (  tool_7_89_present AND tool_6_3_present ) OR  model_present <> 2 THEN
						   loading_status   :='tool not engaged';
						   
					 ELSIF ( tool_6_3_present AND NOT tool_7_89_present) AND  model_present <> 2 THEN
						   loading_Sequence  := 101;
	   
                   END_IF
		    END_IF 
		
		
     60: IF  absoulte_move_done AND SERVO_HME_POS  THEN
     		     servo_move_abs         := FALSE;
     	         loading_Sequence       := 70;
				 
         ELSIF NOT absoulte_move_done AND SERVO_HME_POS THEN 
     			   loading_status   := ' waiting for absolute done ';
     			   
     	 ELSIF 	absoulte_move_done AND NOT SERVO_HME_POS THEN 
     			 loading_status   := ' waiting target pos reached fb ';
     		 
     	 END_IF

     70:  tool_loading_complete:= TRUE;
	      loading_Sequence     := 80;
	 
     80: IF  tool_loading_complete AND tool_unloading_complete THEN
		 unloading_started := FALSE;
		 loading_started   := FALSE;
		 tool_changer_over_complete := TRUE;
		 tool_engagae   := FALSE;
	     END_IF
	  
	  101: IF  operator_ack THEN
		       target_pos_to_servo := target_work_pos ;                                                               
               target_vel_to_servo := target_vel_from_hmi ;
			  IF target_pos_to_servo = target_work_pos AND target_vel_to_servo = target_vel_from_hmi THEN
			     servo_move_abs      := TRUE;
			     loading_status    := ' target position and velocity to servo moved ';
			     loading_Sequence  :=  110;
	         ELSIF target_pos_to_servo <> target_work_pos OR target_vel_to_servo <> target_vel_from_hmi THEN	
		      loading_status   := ' target position or velocity to servo not moved ';
		     END_IF
	     END_IF
	  
	  110: IF absoulte_move_done AND SERVO_WRK_POS  THEN
		     servo_move_abs := FALSE;
			 tool_disengage := TRUE ;
			 disengage_check  := TRUE ;
			 tool_engagae   := FALSE;
			 loading_Sequence  := 120;
			 
		 ELSIF NOT absoulte_move_done AND SERVO_WRK_POS THEN 
			   loading_status   := ' waiting for absolute done ';
	     ELSIF 	absoulte_move_done AND NOT SERVO_WRK_POS THEN 
			 loading_status   := ' waiting target pos reached fb ';		 
		 END_IF 	 
	  
	  120:  IF engage_timer.q THEN
		       target_pos_to_servo := target_work_pos - SERVO_TOL_CHECK_OFFSET_POS;          // moving enage position and velocity to servo                                                     
               target_vel_to_servo := target_vel_from_hmi ;
			   disengage_check       := FALSE;
               IF target_pos_to_servo = target_work_pos- SERVO_TOL_CHECK_OFFSET_POS AND target_vel_to_servo = target_vel_from_hmi THEN
			      servo_move_abs      := TRUE;
			      loading_Sequence  := 130;
			   ELSIF target_pos_to_servo <> target_work_pos- SERVO_TOL_CHECK_OFFSET_POS OR target_vel_to_servo <> target_vel_from_hmi THEN 
				   loading_status   := ' target position or velocity to servo not moved ';
		       END_IF
	        END_IF
			
	  130:  IF NOT (tool_6_3_present AND tool_7_89_present) THEN
		         target_pos_to_servo := target_home_pos;                                                              
                 target_vel_to_servo := target_vel_from_hmi;
			     IF target_pos_to_servo = target_home_pos AND target_vel_to_servo = target_vel_from_hmi THEN
			        servo_move_abs      := TRUE;
			        loading_Sequence  := 140;
				 ELSIF target_pos_to_servo <>  target_home_pos AND target_vel_to_servo <> target_vel_from_hmi THEN  
                       loading_status   := ' target position or velocity to servo not moved '; 
		         END_IF
	        END_IF
			
	 140: 	 IF  absoulte_move_done AND SERVO_HME_POS  THEN
            	     servo_move_abs         := FALSE;
                     loading_Sequence       := 150;
            		 
             ELSIF NOT absoulte_move_done AND SERVO_HME_POS THEN 
            		   loading_status   := ' waiting for absolute done ';
            		   
             ELSIF 	absoulte_move_done AND NOT SERVO_HME_POS THEN 
            		 loading_status   := ' waiting target pos reached fb ';
            	 
             END_IF
			 
      150:   tool_loading_failed := TRUE;
	          
END_CASE


                                                           //////////////////  timer for logic //////////////////////////////// j
														   
disengage_timer(IN:= tool_disengage , PT:= T#5S, Q=> , ET=> );
engage_timer(IN:= engaged_check , PT:= T#5S, Q=> , ET=> );
disengae_timer(IN:= disengage_check , PT:= , Q=> , ET=> );


// #################################	IN RANGE 		##############################


SERVO_WRK_POS		:=In_Range(value:=actual_pos, setvalue:=target_work_pos, tolerance:=0.2 );
SERVO_HME_POS		:=In_Range(value:=actual_pos, setvalue:=target_home_pos, tolerance:=0.2 );
SERVO_TOL_CHCK_POS	:=In_Range(value:=actual_pos, setvalue:=target_work_pos-SERVO_TOL_CHECK_OFFSET_POS, tolerance:=0.2 );

END_FUNCTION_BLOCK

// ---- POUs/Programs/offline testing/servo.TcPOU
FUNCTION_BLOCK servo

VAR_INPUT
	
offline_bit: BOOL;
error_bit: BOOL	;
servo_absolute: BOOL;
target_position: REAL;
servo_pos_delay_time: LTIME;
END_VAR

VAR_OUTPUT
	servo_pos_delay_time_display: LTIME;
	actual_position: REAL;
	absolute_done: BOOL;
END_VAR

VAR
	delay : lton;
	
END_VAR

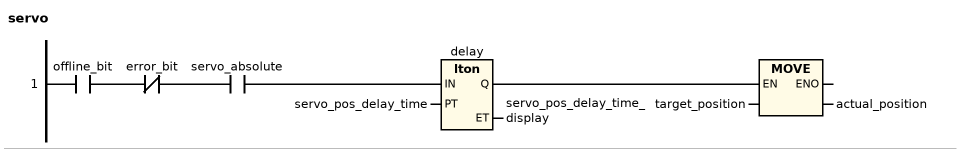
// NETWORK 1
delay(
    IN := offline_bit AND NOT error_bit AND servo_absolute,
    PT := servo_pos_delay_time,
    ET => servo_pos_delay_time_display); // lton
IF delay.Q THEN actual_position := target_position; END_IF

END_FUNCTION_BLOCK

// ---- POUs/Programs/OP50/OP50_MAIN.TcPOU
PROGRAM OP50_MAIN
VAR
	OP50_Modeselection_FB: Mode_Selection_Block1;
	TP_100ms: TP;
	Pulse_1s: BOOL;
	Times: LREAL;
	Pge_NUM : INT;

	Gen_Timer: TON;
END_VAR

OP50_Manual();
OP50_AUTOSEQUENCE();
//OP50_CONVEYOR();
OP50_Camera_FB();
OP50_Error();
OP50_Initialize_Seq();
OP50_Conveyor_Cam_Seq();

//MOdeselection From HMI

IF (OP50_GVL.OP50_HMI_AutoMode AND NOT OP50_GVL.OP50_HMI_ManualMOde AND NOT OP50_GVL.OP50_HMI_StepMode) THEN
	OP50_Modeselection_FB.ModeWord:=1;
	ELSIF (NOT OP50_GVL.OP50_HMI_AutoMode AND OP50_GVL.OP50_HMI_ManualMOde AND NOT OP50_GVL.OP50_HMI_StepMode) THEN
		OP50_Modeselection_FB.ModeWord:=2;
	ELSIF  (NOT OP50_GVL.OP50_HMI_AutoMode AND NOT OP50_GVL.OP50_HMI_ManualMOde AND  OP50_GVL.OP50_HMI_StepMode) THEN
		OP50_Modeselection_FB.ModeWord:=3;
    ELSE   
		OP50_Modeselection_FB.ModeWord:=0;
END_IF

(*
IF  (OP50_AutoSelected OR OP50_ManualSelected ) AND NOT OP50_ErrorActive AND OP50_Safety_OK THEN
  SR50_CONV_servo.bEnable:=TRUE;
  SR50_HORI_servo.bEnable:=TRUE;
  SR50_VERT_servo.bEnable:=TRUE;
ELSE 
  SR50_CONV_servo.bEnable:=FALSE;
  SR50_HORI_servo.bEnable:=FALSE;
  SR50_VERT_servo.bEnable:=FALSE;	
END_IF
*)
IF SR50_CONV_servo.bAxisError OR SR50_HORI_servo.bAxisError OR SR50_VERT_servo.bAxisError THEN
	OP50_ErrorActive:=TRUE;
END_IF
	
OP50_Safety_OK:=OperationEnable;

OP50_Modeselection_FB(
	ModeWord:= , 
	HomeConditionOK:=OP50_HomeConditionOK , 
	OperationEnable:=OP50_AutoSelected AND OP50_Safety_OK , 
	StartPB:=OP50_HMI_Cycle_Start , 
	SafetyAndNOError:= OP50_Safety_OK, 
	ModeAck:=TRUE , 
	HomingINProgress:=OP50_HomeRunning , 
	TempHomeOK:=OP50_Temp_hmeOK , 
	ResetPB:= , 
	AutoSelected=> OP50_AutoSelected, 
	ManualSelected=> OP50_ManualSelected, 
	StepSelected=>OP50_StepSelected , 
	ModeSelAck_Indication=> , 
	StatusDisplay=> , 
	AutoRunning:=OP50_AutoRunning, 
	StepRunning:=OP50_StepRunning , 
	StartEnable:=OP50_StartEnable  , 
	MachineStop:=OP50_Machine_Stop );
	
IF OP50_Stop_Request AND NOT OP50_STN_ENABLE THEN
	OP50_Machine_Stop:=1;
END_IF
Gen_Timer(IN:=OP50_Machine_Stop,PT:=T#5S);
IF Gen_Timer.Q THEN
	OP50_Machine_Stop:=0;
END_IF

END_PROGRAM

// ---- POUs/Programs/OP50/OP50_MANUAL.TcPOU
PROGRAM OP50_MANUAL
VAR
	SR50_Vert_servo_Axis :AXIS_REF;
	SR50_Hori_servo_Axis :AXIS_REF;
	SR50_Conv_servo_Axis :AXIS_REF;
	SR50_GUIDE_GRP_AXIS :AXIS_REF;
	temp_safe: BOOL;
	temp:BOOL;
	OP50_Conveyor	: Servo_Conveyor_FB;
	FESTO_NOT_NEED: BOOL;
	NOT_REQ: BOOL;

	Grip_Test : INT;
	Test : TON;
	b1: BOOL;
	b2: BOOL;
	b3: BOOL;
	b4: BOOL;
	OP50_Camera_Done: BOOL;
	OP50_One_Cycle : BOOL;
	xx: BOOL;
	Conveyor_Track_Delay: TON;
	Conveyor_Track_OFF_Delay: TON;
	Conveyor_Continuous_Run: BOOL;
	Conveyor_Velocity_mode: BOOL;
END_VAR



OP50_VERT_SERVO_POSITION    := SR50_Vert_servo_ctrl.Actual_Position;
OP50_VERT_SERVO_POS_DONE	:= SR50_Vert_servo_ctrl.pos_done ;

OP50_HORI_SERVO_POSITION    := SR50_Hori_servo_ctrl.Actual_Position;
OP50_HORI_SERVO_POS_DONE	:= SR50_Hori_servo_ctrl.pos_done ;

OP50_CONV_SERVO_POSITION    := SR50_CONV_servo_ctrl.Actual_Position;
OP50_CONV_SERVO_POS_DONE	:= SR50_CONV_servo_ctrl.pos_done ;


// VERTICAL SERVO 
IF In_Range(SR50_Vert_servo_status.actualPosition,OP50_VERT_SERVO_SFE_WRK_POS,1) THEN
	OP50_VERT_SERVO_ON_SFE_WRK := TRUE;
ELSE
	OP50_VERT_SERVO_ON_SFE_WRK := FALSE;
END_IF

IF In_Range(SR50_Vert_servo_status.actualPosition,OP50_VERT_SERVO_HME_POS,1) THEN
	OP50_VERT_SERVO_ON_HOME := TRUE;
ELSE
	OP50_VERT_SERVO_ON_HOME := FALSE;
END_IF

IF In_Range(SR50_Vert_servo_status.actualPosition,OP50_VERT_SERVO_PICK_POS,1) THEN
	OP50_VERT_SERVO_ON_WRK_PICK := TRUE;
ELSE
	OP50_VERT_SERVO_ON_WRK_PICK := FALSE;
END_IF		

IF In_Range(SR50_Vert_servo_status.actualPosition,OP50_VERT_SERVO_PLACE_POS,1) THEN
	OP50_VERT_SERVO_ON_WRK_PLACE := TRUE;
ELSE
	OP50_VERT_SERVO_ON_WRK_PLACE := FALSE;
END_IF

//HORIZONTAL SERVO
IF In_Range(SR50_Hori_servo_status.actualPosition,OP50_HORI_SERVO_SFE_WRK_POS,1) THEN
	OP50_HORI_SERVO_ON_SFE_WRK := TRUE;
ELSE
	OP50_HORI_SERVO_ON_SFE_WRK := FALSE;
END_IF

IF In_Range(SR50_Hori_servo_status.actualPosition,OP50_HORI_SERVO_HME_POS,1) THEN
	OP50_HORI_SERVO_ON_HOME := TRUE;
ELSE
	OP50_HORI_SERVO_ON_HOME := FALSE;
END_IF

IF In_Range(SR50_Hori_servo_status.actualPosition,OP50_HORI_SERVO_PICK_POS,4) THEN
	OP50_HORI_SERVO_ON_WRK_PICK := TRUE;
ELSE
	OP50_HORI_SERVO_ON_WRK_PICK := FALSE;
END_IF	

IF In_Range(SR50_Hori_servo_status.actualPosition,OP50_HORI_SERVO_SAFE_PICK_POS,1) THEN
	OP50_HORI_SERVO_ON_SFE_WRK_PICK := TRUE;
ELSE
	OP50_HORI_SERVO_ON_SFE_WRK_PICK := FALSE;
END_IF	

IF In_Range(SR50_Hori_servo_status.actualPosition,OP50_HORI_SERVO_PLACE_POS,1) THEN
	OP50_HORI_SERVO_ON_WRK_PLACE := TRUE;
ELSE
	OP50_HORI_SERVO_ON_WRK_PLACE := FALSE;
END_IF	

//CONVEYOR SERVO

IF In_Range(SR50_CONV_servo_status.actualPosition,OP50_CONV_SERVO_SFE_WRK_POS,1) THEN
	OP50_CONV_SERVO_ON_SFE_WRK := TRUE;
ELSE
	OP50_CONV_SERVO_ON_SFE_WRK := FALSE;
END_IF

IF In_Range(SR50_CONV_servo_status.actualPosition,OP50_CONV_SERVO_HME_POS,1) THEN
	OP50_CONV_SERVO_ON_HOME := TRUE;
ELSE
	OP50_CONV_SERVO_ON_HOME := FALSE;
END_IF

IF In_Range(SR50_CONV_servo_status.actualPosition,OP50_CONV_SERVO_WRK_POS,1) THEN
	OP50_CONV_SERVO_ON_WRK := TRUE;
ELSE
	OP50_CONV_SERVO_ON_WRK := FALSE;
END_IF	


OP50_GVL.SR50_Vert_servo(
	bAxis1_Ref_Switch:= temp, 
	bInit:= , 
	bErrorReset:=OP50_HMI_Reset OR  Servo_Reset, 
	bEnable:=Servo_Enable, 
	bMoveVelocity:= , 
	bHalt:= , 
	bManualMode:= OP50_ManualSelected AND MANUAL_SELECTED ,
	fHomePos:= , 
	fOverride:= , 
	fTargetPosition:=SR50_Vert_servo_ctrl.Position , 
	fTargetVelocity:=SR50_Vert_servo_ctrl.Velocity , 
	fAcc:= , 
	fDec:= ,
	Servo_High_Limit:=OP50_HMI_Vert_High_Limit,
	Servo_Low_Limit:= OP50_HMI_Vert_Low_Limit,	
	WARNING_LIMIT:=1,		
	Actual_Torque=> SR50_Vert_servo_ctrl.Actual_Torque ,
	Actual_position=>SR50_Vert_servo_ctrl.Actual_Position ,
    Actual_velocity=>SR50_Vert_servo_ctrl.Actual_Velocity ,	
	bmove_home:=SR50_Vert_servo_ctrl.Axis_Home_Cmd ,
	baxis_in_home_pos=>SR50_Vert_servo_ctrl.Axis_In_Home ,
	Safe_move_Conditions:=Servo_Safety,
	Axis:= SR50_Vert_servo_Axis , 
	bHome:=SR50_Vert_servo_ctrl.Bsethome ,
	HME_WRITE_ADD:= 16#5009, 
    bSetPosition:=SR50_Vert_servo_ctrl.Bsetpos , 
	bMoveAbsolute:=SR50_Vert_servo_ctrl.ABSmove_Start , 
	bMoveRelative:=SR50_Vert_servo_ctrl.RELmove_Start , 
	bMoveTorque :=SR50_Vert_servo_ctrl.Torque_mode_Start,
	stManualModeAxis:=SR50_Vert_servo_status , 
	sAxisState=>SR50_Vert_servo_ctrl.Axis_State , 
	bAxis_ready=>SR50_Vert_servo_ctrl.Axis_ready , 
	bAxisInPosition=> SR50_Vert_servo_ctrl.Axis_In_Pos, 
	bAxisError=>SR50_Vert_servo_ctrl.Axis_Error , 
	bAxisEnabled=> SR50_Vert_servo_ctrl.Axis_Enabled, 
	bAxisHomed=> SR50_Vert_servo_ctrl.Axis_reference,
	bTorqueReached=> SR50_Vert_servo_ctrl.Trq_reached, 
	bSetPositionDone=>   ,
	bsafe_to_move=> ,
	bABS_Pos_done=> SR50_Vert_servo_ctrl.pos_done , 
	bHaltDone=> , 
	bSTOPDone=> , 
	bHomeDone=> , 
	bDone=> );	

OP50_GVL.SR50_HORI_servo(
	bAxis1_Ref_Switch:= temp, 
	bInit:=temp , 
	bErrorReset:=OP50_HMI_Reset OR Servo_Reset , 
	bEnable:=Servo_Enable , 
	bMoveVelocity:= , 
	bHalt:= , 
	bManualMode:= OP50_ManualSelected AND MANUAL_SELECTED,
	fHomePos:= , 
	fOverride:= , 
	fTargetPosition:= SR50_HORI_servo_ctrl.Position , 
	fTargetVelocity:= SR50_HORI_servo_ctrl.Velocity, 
	fAcc:= , 
	fDec:= ,
	Servo_High_Limit:= OP50_HMI_Hori_High_Limit,	
	Servo_Low_Limit:=  OP50_HMI_Hori_Low_Limit,	 	
	WARNING_LIMIT:=1,	
	Actual_Torque=> SR50_HORI_servo_ctrl.Actual_Torque ,
	Actual_position=>SR50_HORI_servo_ctrl.Actual_Position ,
    Actual_velocity=>SR50_HORI_servo_ctrl.Actual_Velocity ,	
	bmove_home:=SR50_HORI_servo_ctrl.Axis_Home_Cmd ,
	baxis_in_home_pos=>SR50_HORI_servo_ctrl.Axis_In_Home ,
	Safe_move_Conditions:=Servo_Safety,
	Axis:= SR50_HORI_servo_Axis , 
	HME_WRITE_ADD:= 16#5008, 
	bHome:=SR50_HORI_servo_ctrl.Bsethome , 
    bSetPosition:=SR50_HORI_servo_ctrl.Bsetpos , 
	bMoveAbsolute:=SR50_HORI_servo_ctrl.ABSmove_Start , 
	bMoveRelative:=SR50_HORI_servo_ctrl.RELmove_Start , 
	bMoveTorque :=SR50_HORI_servo_ctrl.Torque_mode_Start,
	stManualModeAxis:=SR50_HORI_servo_status , 
	sAxisState=>SR50_HORI_servo_ctrl.Axis_State , 
	bAxis_ready=>SR50_HORI_servo_ctrl.Axis_ready , 
	bAxisInPosition=> SR50_HORI_servo_ctrl.Axis_In_Pos, 
	bAxisError=>SR50_HORI_servo_ctrl.Axis_Error , 
	bAxisEnabled=> SR50_HORI_servo_ctrl.Axis_Enabled, 
	bAxisHomed=> SR50_HORI_servo_ctrl.Axis_reference,
	bTorqueReached=> SR50_HORI_servo_ctrl.Trq_reached, 
	bSetPositionDone=>   ,
	bsafe_to_move=> ,
	bABS_Pos_done=> SR50_HORI_servo_ctrl.pos_done , 
	bHaltDone=> , 
	bSTOPDone=> , 
	bHomeDone=> , 
	bDone=> );

CASE Grip_Test OF
	1: IF Test.Q AND NOT  SR50_HORI_servo_ctrl.ABSmove_Start THEN
		SR50_HORI_servo_ctrl.Position:=1;
	    SR50_HORI_servo_ctrl.ABSmove_Start:=1;
	    Grip_Test:=2;
	   END_IF	
	   
	2: IF Test.Q AND NOT SR50_HORI_servo_ctrl.ABSmove_Start THEN
		SR50_HORI_servo_ctrl.Position:=200;
		SR50_HORI_servo_ctrl.ABSmove_Start:=1;
		Grip_Test:=1;
	   END_IF	  
END_CASE

Test(IN:= NOT SR50_HORI_servo_ctrl.ABSmove_Start , PT:=T#500MS);	
	
	
	
	
SR50_CONV_servo(
	bAxis1_Ref_Switch:= temp, 
	bInit:= , 
	bErrorReset:=OP50_HMI_Reset OR Servo_reset , 
	bEnable:=Servo_Enable, 
	bMoveVelocity:=SR50_CONV_servo_ctrl.VELmove_Start , 
	bHalt:= , 
	bManualMode:= OP50_ManualSelected and MANUAL_SELECTED,
	fHomePos:= , 
	fOverride:= , 
	fTargetPosition:= SR50_CONV_servo_ctrl.Position, 
	fTargetVelocity:= SR50_CONV_servo_ctrl.Velocity, 
	LIMIT_BYPASS:=1,
	fAcc:= , 
	fDec:= ,
	Actual_Torque=> SR50_CONV_servo_ctrl.Actual_Torque ,
	Actual_position=>SR50_CONV_servo_ctrl.Actual_Position ,
    Actual_velocity=>SR50_CONV_servo_ctrl.Actual_Velocity ,	
	bmove_home:=SR50_CONV_servo_ctrl.Axis_Home_Cmd ,
	baxis_in_home_pos=>SR50_CONV_servo_ctrl.Axis_In_Home ,
	Safe_move_Conditions:=Servo_safety,
	Axis:= SR50_CONV_servo_Axis , 
	HME_WRITE_ADD:= 16#500A,	
	bHome:=SR50_CONV_servo_ctrl.Bsethome , 
    bSetPosition:=SR50_CONV_servo_ctrl.Bsetpos , 
	bMoveAbsolute:=SR50_CONV_servo_ctrl.ABSmove_Start , 
	bMoveRelative:=SR50_CONV_servo_ctrl.RELmove_Start , 
	bMoveTorque :=SR50_CONV_servo_ctrl.Torque_mode_Start,
	stManualModeAxis:=SR50_CONV_servo_status , 
	sAxisState=>SR50_CONV_servo_ctrl.Axis_State , 
	bAxis_ready=>SR50_CONV_servo_ctrl.Axis_ready , 
	bAxisInPosition=> SR50_CONV_servo_ctrl.Axis_In_Pos, 
	bAxisError=>SR50_CONV_servo_ctrl.Axis_Error , 
	bAxisEnabled=> SR50_CONV_servo_ctrl.Axis_Enabled, 
	bAxisHomed=> SR50_CONV_servo_ctrl.Axis_reference,
	bTorqueReached=> SR50_CONV_servo_ctrl.Trq_reached, 
	bSetPositionDone=>   ,
	bsafe_to_move=>SR50_CONV_servo_ctrl.Safe_To_Move ,
	bABS_Pos_done=> SR50_CONV_servo_ctrl.pos_done , 
	bHaltDone=> , 
	bSTOPDone=> , 
	bHomeDone=> , 
	bDone=> );	
	
IF OP50_ManualSelected OR MANUAL_SELECTED THEN
	SR50_Vert_servo_status.targetVelocity:=10;
	SR50_Hori_servo_status.targetVelocity:=10;
END_IF

//LH Rejection Cylinder
//move ZERO to STATUS
//CR50_LH_Rej_Cyl_Status:=0;

//Reset Auto Cmd IN Manual Mode & Homing
IF (OP50_Auto OR OP50_HomeRunning) THEN
	CR50_LH_Rej_Cyl.AutoCmd1:=FALSE;
	CR50_LH_Rej_Cyl.AutoCmd2:=FALSE;		
END_IF

// Safe Home
IF (TRUE) AND  (TRUE) THEN 
	CR50_LH_Rej_Cyl.SafeHome:= TRUE ;
ELSE 
	CR50_LH_Rej_Cyl.SafeHome:= FALSE ;
END_IF
// Safe Work
IF (TRUE) OR (TRUE) THEN 
	CR50_LH_Rej_Cyl.Safework:= TRUE ;
ELSE 
	CR50_LH_Rej_Cyl.Safework:= FALSE ;
END_IF
	
// Manual PB  Cyl Mapping
IF (OP50_HMI_LH_Rej_Cyl_Home_PB=TRUE) THEN
	CR50_LH_Rej_Cyl.ManualPB1:=TRUE;
ELSE 
	CR50_LH_Rej_Cyl.ManualPB1:=FALSE;
END_IF
	
IF (OP50_HMI_LH_Rej_Cyl_Work_PB=TRUE) THEN
	CR50_LH_Rej_Cyl.ManualPB2:=TRUE;
ELSE 
	CR50_LH_Rej_Cyl.ManualPB2:=FALSE;
END_IF
	
CR50_LH_Rej_Cyl(
	Auto:= OP50_AutoSelected , 
	Manual:= OP50_ManualSelected AND MANUAL_SELECTED, 
	ErrorActive:= , 
	ResetPB:= OP50_HMI_Reset, 
	Sensor1:= I50_LH_REJ_CYL_FWD_I1101_2, 
	Sensor2:= I50_LH_REJ_CYL_REV_I1101_3,
	ManualPB1:= , 
	ManualPB2:= , 
	AutoCmd1:= , 
	AutoCmd2:= , 
	OperationEnable:= OperationEnable , 
	SafeHome:= , 
	SafeWork:= , 
	HomingCmd1:= , 
	Pulse_1Sec:= Pulse_Block.Q1Hz , 
	BlinkingBit:= , 
	TimeOut1:= 5, 
	TimeOut2:= 5, 
	TimeOut3:= 5, 
	Solenoid1=>  O50_LH_REJ_CYL_FWD_Q1151_7, 
	Solenoid2=>  O50_LH_REJ_CYL_REV_Q1151_6,
	AlarmSensor1=> , 
	AlarmSensor2=> , 
	AlarmSolenoid1=> , 
	AlarmSolenoid2=> , 
	AllSignal=> , 
	AlarmPresent=> , 
	Position1=> , 
	Position2=> , 
	HomeSensorBlink=> , 
	WorkSensorBlink=> , 
	Status:=CR50_LH_Rej_Cyl_status );


//RH Rejection Cylinder
//move ZERO to STATUS
//CR50_RH_Rej_Cyl_Status:=0;

//Reset Auto Cmd IN Manual Mode & Homing
IF (OP50_Auto OR OP50_HomeRunning) THEN
	CR50_RH_Rej_Cyl.AutoCmd1:=FALSE;
	CR50_RH_Rej_Cyl.AutoCmd2:=FALSE;		
END_IF

// Safe Home
IF (TRUE) AND  (TRUE) THEN 
	CR50_RH_Rej_Cyl.SafeHome:= TRUE ;
ELSE 
	CR50_RH_Rej_Cyl.SafeHome:= FALSE ;
END_IF
// Safe Work
IF (TRUE) OR (TRUE) THEN 
	CR50_RH_Rej_Cyl.Safework:= TRUE ;
ELSE 
	CR50_RH_Rej_Cyl.Safework:= FALSE ;
END_IF
	
// Manual PB  Cyl Mapping
IF (OP50_HMI_RH_Rej_Cyl_Home_PB=TRUE) THEN
	CR50_RH_Rej_Cyl.ManualPB1:=TRUE;
ELSE 
	CR50_RH_Rej_Cyl.ManualPB1:=FALSE;
END_IF
	
IF (OP50_HMI_RH_Rej_Cyl_Work_PB=TRUE) THEN
	CR50_RH_Rej_Cyl.ManualPB2:=TRUE;
ELSE 
	CR50_RH_Rej_Cyl.ManualPB2:=FALSE;
END_IF
	
CR50_RH_Rej_Cyl(
	Auto:= OP50_AutoSelected ,  
	Manual:= OP50_ManualSelected AND MANUAL_SELECTED, 
	ErrorActive:= , 
	ResetPB:= OP50_HMI_Reset,                    
	Sensor1:= I50_RH_REJ_CYL_FWD_I1101_4 , 
	Sensor2:= I50_RH_REJ_CYL_REV_I1101_5 , 
	ManualPB1:= , 
	ManualPB2:= , 
	AutoCmd1:= , 
	AutoCmd2:= , 
	OperationEnable:= OperationEnable, 
	SafeHome:= , 
	SafeWork:= , 
	HomingCmd1:= , 
	Pulse_1Sec:= Pulse_Block.Q1Hz , 
	BlinkingBit:= , 
	TimeOut1:= 5, 
	TimeOut2:= 5, 
	TimeOut3:= 5, 
	Solenoid1=> O50_RH_REJ_CYL_FWD_Q1152_1 , 
	Solenoid2=> O50_RH_REJ_CYL_REV_Q1152_0 , 
	AlarmSensor1=> , 
	AlarmSensor2=> , 
	AlarmSolenoid1=>, 
	AlarmSolenoid2=> , 
	AllSignal=> , 
	AlarmPresent=> , 
	Position1=> , 
	Position2=> , 
	HomeSensorBlink=> , 
	WorkSensorBlink=> , 
	Status:=CR50_RH_Rej_Cyl_status );	
	
OP50_GIUDE_GRP_ctrl.Velocity:=50;	
	
OP50_GIUDE_GRP(														// FESTO GUIDE GRIPPER
	bAxis1_Ref_Switch:= , 
	bInit:=  , 
	bErrorReset:= Servo_Reset , 
	bEnable:= Servo_Enable , /// MACHINE ERR REGISTER CHANGE
	bMoveVelocity:= , 
	bHalt:= , 
	bManualMode:= OP50_ManualSelected AND MANUAL_SELECTED , 									//MANUAL REGISTER CHANGE
	fHomePos:= , 
	fOverride:= , 
	fTargetPosition:= OP50_GIUDE_GRP_ctrl.Position, 
	fTargetVelocity:= OP50_GIUDE_GRP_ctrl.Velocity, 
	fAcc:= , 
	fDec:= , 
	Servo_High_Limit:= 100,	
	Servo_Low_Limit:= -100,	 	
	WARNING_LIMIT:=1,		
	Safe_move_Conditions:= Servo_Safety,
	TORQUE_APPLIED :=  , 					// CHANGE
	Axis:= SR50_GUIDE_GRP_AXIS, 
	bHome:= OP50_GIUDE_GRP_ctrl.Bsethome, 
	bSetPosition:= FESTO_NOT_NEED , 
	bMoveAbsolute:= OP50_GIUDE_GRP_ctrl.ABSmove_Start,
	bMoveRelative:= NOT_REQ , 
	bMoveTorque:= NOT_REQ , 
	stManualModeAxis:= OP50_GIUDE_GRP_Manual_Axis, 
 	sAxisState=>OP50_GIUDE_GRP_ctrl.Axis_State , 
	baxis_in_home_pos=>OP50_GIUDE_GRP_ctrl.Axis_In_Home ,
	bAxis_ready=> , 
	bAxisInPosition=> , 
	bAxisError=> , 
	bAxisEnabled=> , 
	bAxisHomed=> , 
	bSetPositionDone=> , 
	bHaltDone=> , 
	bSTOPDone=> , 
	bHomeDone=>OP50_GIUDE_GRP_ctrl.Axis_Home_Done , 
	bDone=> , 
	bTorqueReached=> , 
	bsafe_to_move=> , 
	baxis_in_home_pos=> , 
	bABS_Pos_done=> OP50_GIUDE_GRP_ctrl.Axis_In_Pos, 
	Actual_position=>OP50_GIUDE_GRP_ctrl.Actual_Position,
	Actual_velocity=>OP50_GIUDE_GRP_ctrl.Actual_Velocity , 
	Actual_Torque=> );
	
OP50_GIUDE_GRP_Manual_Axis.targetVelocity := 50;	
//LH Gripper Cylinder
//move ZERO to STATUS
//CR50_LH_Grip_Cyl_Status:=0;

//Reset Auto Cmd IN Manual Mode & Homing
//IF (OP50_Auto OR OP50_HomeRunning) THEN
//	CR50_LH_Grip_Cyl.AutoCmd1:=FALSE;
//	CR50_LH_Grip_Cyl.AutoCmd2:=FALSE;		
//END_IF

// Safe Home
IF (TRUE) AND  (TRUE) THEN 
	CR50_LH_Grip_Cyl.SafeHome:= TRUE ;
ELSE 
	CR50_LH_Grip_Cyl.SafeHome:= FALSE ;
END_IF
// Safe Work
IF (TRUE) OR (TRUE) THEN 
	CR50_LH_Grip_Cyl.Safework:= TRUE ;
ELSE 
	CR50_LH_Grip_Cyl.Safework:= FALSE ;
END_IF
	
// Manual PB  Cyl Mapping
IF (OP50_HMI_LH_Grip_Cyl_Home_PB=TRUE) THEN
	CR50_LH_Grip_Cyl.ManualPB1:=TRUE;
ELSE 
	CR50_LH_Grip_Cyl.ManualPB1:=FALSE;
END_IF
	
IF (OP50_HMI_LH_Grip_Cyl_Work_PB=TRUE) THEN
	CR50_LH_Grip_Cyl.ManualPB2:=TRUE;
ELSE 
	CR50_LH_Grip_Cyl.ManualPB2:=FALSE;
END_IF
	
CR50_LH_Grip_Cyl(
	Auto:= OP50_AutoSelected , 
	Manual:= OP50_ManualSelected AND MANUAL_SELECTED, 
	ErrorActive:= , 
	ResetPB:= OP50_HMI_Reset, 
	Sensor1:=I50_LH_GRIP_CLSE_I1101_7 , 
	Sensor2:=NOT I50_LH_GRIP_CLSE_I1101_7 ,
	ManualPB1:= , 
	ManualPB2:= , 
	AutoCmd1:= , 
	AutoCmd2:= , 
	OperationEnable:= OperationEnable , 
	SafeHome:= , 
	SafeWork:= , 
	HomingCmd1:= , 
	Pulse_1Sec:= Pulse_Block.Q1Hz , 
	BlinkingBit:= , 
	TimeOut1:= 5, 
	TimeOut2:= 5, 
	TimeOut3:= 5, 
	Solenoid1=> O50_LH_GRIP_CLSE_Q1151_3  , 
	Solenoid2=> O50_LH_GRIP_OPN_Q1151_2  ,
	AlarmSensor1=> , 
	AlarmSensor2=> , 
	AlarmSolenoid1=> , 
	AlarmSolenoid2=> , 
	AllSignal=> , 
	AlarmPresent=> , 
	Position1=> , 
	Position2=> , 
	HomeSensorBlink=> , 
	WorkSensorBlink=> , 
	Status:=CR50_LH_Grip_Cyl_status );
	
//RH Gripection Cylinder
//move ZERO to STATUS
//CR50_RH_Grip_Cyl_Status:=0;

//Reset Auto Cmd IN Manual Mode & Homing
//IF (OP50_Auto OR OP50_HomeRunning) THEN
//	CR50_RH_Grip_Cyl.AutoCmd1:=FALSE;
//	CR50_RH_Grip_Cyl.AutoCmd2:=FALSE;		
//END_IF

// Safe Home
IF (TRUE) AND  (TRUE) THEN 
	CR50_RH_Grip_Cyl.SafeHome:= TRUE ;
ELSE 
	CR50_RH_Grip_Cyl.SafeHome:= FALSE ;
END_IF
// Safe Work
IF (TRUE) OR (TRUE) THEN 
	CR50_RH_Grip_Cyl.Safework:= TRUE ;
ELSE 
	CR50_RH_Grip_Cyl.Safework:= FALSE ;
END_IF
	
// Manual PB  Cyl Mapping
IF (OP50_HMI_RH_Grip_Cyl_Home_PB=TRUE) THEN
	CR50_RH_Grip_Cyl.ManualPB1:=TRUE;
ELSE 
	CR50_RH_Grip_Cyl.ManualPB1:=FALSE;
END_IF
	
IF (OP50_HMI_RH_Grip_Cyl_Work_PB=TRUE) THEN
	CR50_RH_Grip_Cyl.ManualPB2:=TRUE;
ELSE 
	CR50_RH_Grip_Cyl.ManualPB2:=FALSE;
END_IF
	
CR50_RH_Grip_Cyl(
	Auto:= OP50_AutoSelected , 
	Manual:= OP50_ManualSelected OR MANUAL_SELECTED, 
	ErrorActive:= , 
	ResetPB:= OP50_HMI_Reset, 
	Sensor1:= I50_RH_GRIP_CLSE_I1110_1, 
	Sensor2:= NOT I50_RH_GRIP_CLSE_I1110_1,
	ManualPB1:= , 
	ManualPB2:= , 
	AutoCmd1:= , 
	AutoCmd2:= , 
	OperationEnable:= OperationEnable , 
	SafeHome:= , 
	SafeWork:= , 
	HomingCmd1:= , 
	Pulse_1Sec:= Pulse_Block.Q1Hz , 
	BlinkingBit:= , 
	TimeOut1:= 5, 
	TimeOut2:= 5, 
	TimeOut3:= 5, 
	Solenoid1=> O50_RH_GRIP_CLSE_Q1151_5 , 
	Solenoid2=> O50_RH_GRIP_OPN_Q1151_4,
	AlarmSensor1=> , 
	AlarmSensor2=> , 
	AlarmSolenoid1=> , 
	AlarmSolenoid2=> , 
	AllSignal=> , 
	AlarmPresent=> , 
	Position1=> , 
	Position2=> , 
	HomeSensorBlink=> , 
	WorkSensorBlink=> , 
	Status:=CR50_RH_Grip_Cyl_status );

IF OP50_Gripper_LH_Open AND NOT OP50_HomeRunning THEN
 CR50_LH_Grip_Cyl.AutoCmd2:=1;
 CR50_LH_Grip_Cyl.AutoCmd1:=0;
 IF NOT I50_LH_GRIP_CLSE_I1101_7 THEN
   OP50_Gripper_LH_State:=1;
   OP50_Gripper_LH_Open:=0;
 END_IF
END_IF 

IF OP50_Gripper_LH_Close AND NOT OP50_HomeRunning THEN
 CR50_LH_Grip_Cyl.AutoCmd1:=1;
 CR50_LH_Grip_Cyl.AutoCmd2:=0;
 IF NOT I50_LH_GRIP_CLSE_I1101_7 THEN
   OP50_Gripper_LH_State:=0;
   OP50_Gripper_LH_Close:=0;
 END_IF 
END_IF 

IF OP50_Gripper_RH_Open AND NOT OP50_HomeRunning THEN
  OP50_Gripper_RH_Close:=0;
  CR50_RH_Grip_Cyl.AutoCmd2:=1;
  CR50_RH_Grip_Cyl.AutoCmd1:=0;
  if not I50_RH_GRIP_CLSE_I1110_1 THEN
   OP50_Gripper_RH_State:=1;
   OP50_Gripper_RH_Open:=0;
  END_IF 
END_IF 

IF OP50_Gripper_RH_Close AND NOT OP50_HomeRunning THEN
 OP50_Gripper_RH_Open:=0;
 CR50_RH_Grip_Cyl.AutoCmd1:=1;
 CR50_RH_Grip_Cyl.AutoCmd2:=0;
 if not I50_RH_GRIP_CLSE_I1110_1 THEN
   OP50_Gripper_RH_State:=0;
   OP50_Gripper_RH_Close:=0;
 END_IF 
END_IF 
	
IF OP50_ManualSelected OR OP50_HomeRunning THEN
  CR50_LH_Grip_Cyl.AutoCmd1:=0;
  CR50_LH_Grip_Cyl.AutoCmd2:=0;	
  CR50_RH_Grip_Cyl.AutoCmd2:=0;
  CR50_RH_Grip_Cyl.AutoCmd1:=0;
END_IF

END_PROGRAM

// ---- POUs/Programs/OP50/OP50_CONVEYOR.TcPOU
PROGRAM OP50_CONVEYOR
VAR
	con_step_no : INT;
	cam_trig : BOOL;
	cam_ok : BOOL;
	LH_Cam_OK : BOOL;
	RH_Cam_OK : BOOL;
	go : BOOL;
	t1: ton;
	t2: ton;
	t3: ton;
	t4: ton;
	
	temp: BOOL;
	check:BOOL;
	check1:ton;
	fwd_time : INT :=500;
	rev_time : INT :=500;
	count_nok :INT;
	forward: BOOL;
	reverse: BOOL;
		temp_3 : BOOl;
END_VAR

IF (NOT OP50_AutoSelected OR OP50_ErrorActive ) THEN
	SR50_CONV_servo_ctrl.VELmove_Start:=FALSE;
	forward:=FALSE;
	reverse:=FALSE;
	con_step_no:= 10;
END_IF	

OP50_Model:=Model;


IF MANUAL_SELECTED AND OP50_ManualSelected THEN               
	IF I50_DRUM_CONV_REV_I306_3 THEN
		SR50_Conv_servo_status.targetVelocity:=OP50_Conv_Rev_Speed_6_3;
		SR50_CONV_servo_ctrl.VELmove_Start:=I50_DRUM_CONV_REV_I306_3;
 	ELSIF I50_DRUM_CONV_FWD_I306_4 THEN
		SR50_Conv_servo_status.targetVelocity:=OP50_Conv_Fwd_Speed_7_89;
		SR50_CONV_servo_ctrl.VELmove_Start:=I50_DRUM_CONV_FWD_I306_4;	
	ELSE 	
		SR50_CONV_servo_ctrl.VELmove_Start:=0;   	
	END_IF  	
END_IF
             
IF OP50_Model='6.3' THEN
	fwd_time:=OP50_Conv_Fwd_Time_6_3;
	rev_time:=OP50_Conv_Rev_Time_6_3;
	IF forward THEN
		OP50_Conveyor_Speed:=OP50_Conv_Fwd_Speed_6_3;
	END_IF
	IF reverse THEN
		OP50_Conveyor_Speed:=OP50_Conv_Rev_Speed_6_3;
	END_IF
END_IF

IF OP50_Model='7.89' THEN
	fwd_time:=OP50_Conv_Fwd_Time_7_89;
	rev_time:=OP50_Conv_Rev_Time_7_89;
	IF forward THEN
		OP50_Conveyor_Speed:=OP50_Conv_Fwd_Speed_7_89;
	END_IF
	IF reverse THEN
		OP50_Conveyor_Speed:=OP50_Conv_Rev_Speed_7_89;
	END_IF
END_IF

CASE con_step_no OF
		10: IF (OP50_AutoSelected) THEN		// Check Automode Selected
				con_step_no:=65;
	        END_IF
		   
        65:	SR50_CONV_servo_ctrl.Velocity:= OP50_Conveyor_Speed;		
			forward:=TRUE;
			SR50_CONV_servo_ctrl.VELmove_Start:=TRUE;	
			IF t2.Q THEN
    			forward:=FALSE;
				SR50_CONV_servo_ctrl.VELmove_Start:=FALSE;
				con_step_no:= 70;
			END_IF
		  
		70: IF NOT SR50_CONV_servo_ctrl.VELmove_Start THEN
			  cam_trig :=TRUE;
			  IF t1.Q THEN
				con_step_no:= 75;
			  END_IF
			END_IF	
					
		75:	IF cam_ok AND NOT SR50_CONV_servo_ctrl.VELmove_Start AND SR50_CONV_servo_ctrl.Axis_ready THEN
				IF LH_Cam_OK AND RH_Cam_OK THEN
				 con_step_no:= 90;
				 fwd_time:=OP50_Conv_Fwd_Time_6_3;
				 count_nok:=0;	
				ELSIF (NOT LH_Cam_OK OR NOT RH_Cam_OK) AND count_nok<5 THEN
				 count_nok := count_nok +1;
				 con_step_no:= 76;	
				ELSIF count_nok>=5 THEN
	             fwd_time:=5000;
				 con_step_no:= 80; 
				END_IF
			END_IF	
			
		76:	 IF NOT LH_Cam_OK AND NOT SR50_CONV_servo_ctrl.VELmove_Start THEN
				CR50_LH_Rej_Cyl.AutoCmd2:=TRUE;
				IF  I50_LH_REJ_CYL_FWD_I1101_2  THEN
					CR50_LH_Rej_Cyl.AutoCmd1:=1;
					CR50_LH_Rej_Cyl.AutoCmd2:=0;					
				END_IF
				IF I50_LH_REJ_CYL_REV_I1101_3 AND count_nok<5 AND NOT CR50_LH_Rej_Cyl.AutoCmd2 THEN
					CR50_LH_Rej_Cyl.AutoCmd2:=0;
					fwd_time:=OP50_Conv_Fwd_Time_6_3;
				    con_step_no:= 77;
				END_IF
                IF count_nok>5 THEN
					fwd_time:=5000;
				    con_step_no:= 77;	
				END_IF
			ELSIF LH_Cam_OK THEN
				con_step_no:= 77;
			END_IF	
			
	   77:	IF NOT RH_Cam_OK AND NOT SR50_CONV_servo_ctrl.VELmove_Start THEN	
				CR50_RH_Rej_Cyl.AutoCmd2:=TRUE;
				IF  I50_RH_REJ_CYL_FWD_I1101_4 THEN
					CR50_RH_Rej_Cyl.AutoCmd1:=1;
					CR50_RH_Rej_Cyl.AutoCmd2:=0;				
				END_IF
				IF I50_RH_REJ_CYL_REV_I1101_5 AND count_nok<5 AND NOT CR50_RH_Rej_Cyl.AutoCmd2 THEN
					CR50_RH_Rej_Cyl.AutoCmd2:=0;					
					fwd_time:=OP50_Conv_Fwd_Time_6_3;
				    con_step_no:= 80;
				END_IF
				IF count_nok>5 THEN
					fwd_time:=5000;
				    con_step_no:= 80;	
				END_IF
			ELSIF RH_Cam_OK THEN
				con_step_no:= 80;
			END_IF		
			
		80: 	IF fwd_time=5000 THEN
			       count_nok:=0;	
				END_IF
                SR50_CONV_servo_ctrl.Velocity:= OP50_Conveyor_Speed;				
				forward:=TRUE;
				SR50_CONV_servo_ctrl.VELmove_Start:=TRUE;	
				IF t2.Q THEN
    				forward:=FALSE;
					SR50_CONV_servo_ctrl.VELmove_Start:=FALSE;
					con_step_no:= 70;
				END_IF
		        
		90: 	SR50_CONV_servo_ctrl.Velocity:= OP50_Conveyor_Speed;
				reverse:=TRUE;
				SR50_CONV_servo_ctrl.VELmove_Start:=TRUE;
				IF t3.Q THEN
 					reverse:=FALSE;
					SR50_CONV_servo_ctrl.VELmove_Start:=FALSE;
					con_step_no:= 100;
				END_IF		
				
		100: OP50_pick_ready:=TRUE;
			 IF OP50_pick_done or temp_3 THEN
				 OP50_pick_ready :=FALSE;
				 OP50_pick_done:=FALSE;
				 con_step_no:= 80;
			 END_IF
			 		
				
END_CASE

t1(IN:=cam_trig ,PT:=T#500MS);
IF cam_trig AND con_step_no=70  THEN
	cam_ok:=FALSE;
END_IF
IF t1.Q THEN
	LH_Cam_OK:=1;
	RH_Cam_OK:=1;
	cam_ok:=temp;
	cam_trig :=FALSE;
END_IF

t2(IN:=forward ,PT:=INT_TO_TIME(fwd_time));
t3(IN:=reverse ,PT:=INT_TO_TIME(rev_time));
t4(IN:=cam_ok,PT:=T#1S);

END_PROGRAM

// ---- POUs/Programs/OP50/OP50_AUTOSEQUENCE.TcPOU
PROGRAM OP50_AUTOSEQUENCE
VAR
	OP50_Oring_OK 	: BOOL;
	FIXTURE_LH		: INT;
	FIXTURE_RH 		: INT;
	del : ton;
	tmp :BOOL;
	Gripper_Delay  			: TON;
	Gripper_pick_Delay		: TON;
	Gripper_Aft_pick_Delay  : TON;
	Gripper_Place_Delay		: TON;
	Gripper_Aft_Place_Delay	: TON;
	Rejection_Grip_Delay	: TON;	
	OP50_STN_MOVER: INT;
	Dry_run : BOOL;
	
	PAP_CYC_VAR : BOOL;
	OP50_PAP_Cycle_time : UDINT;
	OP50_Overall_Cyc_Time	: UDINT;
	OP50_Cycle_Time_FB : FB_Cycletime;
	OP50_PAP_Cycle_Time_FB : FB_Cycletime;
	OP50_Continous_Run : BOOL;
	
END_VAR

// AUTO MODE
IF (NOT OP50_AutoSelected OR  OP50_ErrorActive OR OP50_HomeRunning ) THEN
	OP50_AutoRunning:= FALSE;
	OP50_AutoSeq:= 10;
END_IF	

IF OP50_AutoSelected THEN
	OP50_GIUDE_GRP_ctrl.Position:=OP50_Guide_Pos;
	OP50_GIUDE_GRP_ctrl.Velocity:=50;	
	SR50_Vert_servo_ctrl.Velocity:=OP50_HMI_Servo_Speed_Vertical;
	SR50_HORI_servo_ctrl.Velocity:=OP50_HMI_Servo_Speed_Horizontal;	
END_IF

IF NOT OP50_AutoRunning THEN
    OP50_GIUDE_GRP_ctrl.Position:=0;
	OP50_GIUDE_GRP_ctrl.Velocity:=50;
	IF NOT In_Range(OP50_GIUDE_GRP_ctrl.Actual_Position,0,0.5) THEN
		OP50_GIUDE_GRP_ctrl.ABSmove_Start:=TRUE;
	END_IF	
END_IF

CASE OP50_AutoSeq OF
	    10: IF (OP50_AutoSelected) THEN		// Check Automode Selected
				OP50_AutoSeq:=20;
	        END_IF
		
	    20:IF (NOT OP50_ErrorActive) THEN		//Check No error
		       OP50_AutoSeq:=30;
      	   END_IF
		   
      	30:IF (NOT OP50_HomeRunning) THEN		//Check No Homerunning
      		   OP50_AutoSeq :=40;
      	   END_IF
		   
        40:IF (OP50_Main.OP50_Modeselection_FB.TempHomeOK)THEN	//Check Machine in Home
      		   OP50_AutoSeq:= 50;
      	   END_IF
		   
      	50:IF ( NOT OP50_OperationCompleted) THEN		// Check Operation Completed Reset
      		   OP50_AutoSeq:=60;
      	   END_IF
		   
		60:IF  ( OP50_AutoRunning OR (NOT OP50_AutoRunning AND OP50_HMI_Cycle_Start )) THEN		//Machine Start in Fully Automatic or Press Cycle Start For Semi Automatic
		    OP50_GVL.OP50_HomeConditionOK:=TRUE;
	 			IF( OP50_Main.OP50_Modeselection_FB.HomeConditionOK AND OP50_AutoSelected) THEN
					OP50_GVL.OP50_AutoRunning:=TRUE;
					OP50_GVL.OP50_StepRunning:= FALSE;				
				ELSIF (OP50_Main.OP50_Modeselection_FB.HomeConditionOK AND OP50_StepSelected) THEN
					OP50_GVL.OP50_AutoRunning:=FALSE;
					OP50_GVL.OP50_StepRunning:= TRUE;
				END_IF;
		  END_IF
		   IF ((OP50_AutoRunning OR OP50_StepRunning) AND OP50_StartEnable) THEN
			   OP50_GIUDE_GRP_ctrl.ABSmove_Start:=TRUE;
			   OP50_AutoSeq:= 65;
		   END_IF	
		
	    65 :  OP50_Gripper_LH_Close:=TRUE;  //CHECKING GRIPPER STATE BEFORE GRIPPING
			  OP50_Gripper_RH_Close:=TRUE;
			  IF NOT OP50_Gripper_LH_State AND NOT OP50_Gripper_RH_State THEN
				   OP50_AutoSeq:=66;
			  ELSE 	   
				   OP50_AutoSeq:=220;
			  END_IF    
		   
	    66: PAP_CYC_VAR:=1;
			IF OP50_pick_ready THEN
				OP50_AutoSeq:=70;
			ELSE 
				OP50_AutoSeq:=86;	
			END_IF 
		   
		70 : //MOVING HORIZONTAL SERVO TO PICK POSITION
			  IF (OP50_HORI_SERVO_ON_SFE_WRK OR OP50_HORI_SERVO_ON_HOME OR OP50_HORI_SERVO_ON_WRK_PLACE OR OP50_HORI_SERVO_ON_WRK_PICK )AND OP50_HORI_SERVO_POS_DONE AND NOT SR50_HORI_servo_ctrl.ABSmove_Start THEN 
			   SR50_Hori_servo_ctrl.Position:=OP50_HORI_SERVO_PICK_POS;
               OP50_AutoSeq:=80;		  
	          END_IF
			 
		80 :  SR50_HORI_servo_ctrl.ABSmove_Start := TRUE;     //HORIZONTAL SERVO MOVING
		       IF OP50_HORI_SERVO_ON_WRK_PICK THEN
				   SR50_HORI_servo_ctrl.ABSmove_Start := FALSE;
				   IF OP50_Gripper_LH_State AND OP50_Gripper_RH_State THEN
				        OP50_AutoSeq:=85;
				   ELSE 
						OP50_AutoSeq:=82;
				   END_IF
			   END_IF
		
	  	82 :  OP50_Gripper_LH_Close:=TRUE;  //CHECKING GRIPPER STATE BEFORE GRIPPING
			  OP50_Gripper_RH_Close:=TRUE;
			  IF NOT OP50_Gripper_LH_State AND NOT OP50_Gripper_RH_State THEN
				   OP50_AutoSeq:=85;
			  END_IF
			   
		85:	   // MOVING VERTICAL SERVO TO PICK POSITION
               IF OP50_HORI_SERVO_ON_WRK_PICK AND (OP50_VERT_SERVO_ON_SFE_WRK OR OP50_VERT_SERVO_ON_HOME) AND 
				   OP50_VERT_SERVO_POS_DONE AND NOT SR50_VERT_servo_ctrl.ABSmove_Start  THEN
				   SR50_Vert_servo_ctrl.Position:=OP50_VERT_SERVO_PICK_POS;
				   SR50_VERT_servo_ctrl.ABSmove_Start := TRUE;
              	   OP50_AutoSeq:=100;			   
			   END_IF

	    86:   IF (OP50_HORI_SERVO_ON_SFE_WRK OR OP50_HORI_SERVO_ON_HOME OR OP50_HORI_SERVO_ON_WRK_PLACE OR OP50_HORI_SERVO_ON_WRK_PICK )AND OP50_HORI_SERVO_POS_DONE AND NOT SR50_HORI_servo_ctrl.ABSmove_Start THEN 
			    SR50_Hori_servo_ctrl.Position:=OP50_HORI_SERVO_SAFE_PICK_POS;
			    SR50_HORI_servo_ctrl.ABSmove_Start := TRUE;
                OP50_AutoSeq:=90;
			  END_IF
			   		  
		90 : IF OP50_pick_ready THEN  // WAITING FOR O-RING TO BE OK AND THEN MOVING THE VERTICAL SERVO
			 	SR50_Hori_servo_ctrl.Position:=OP50_HORI_SERVO_PICK_POS;
				SR50_Hori_servo_ctrl.ABSmove_Start := TRUE;
				OP50_AutoSeq:=92;
		     END_IF				  				

		92: SR50_Hori_servo_ctrl.ABSmove_Start := TRUE;
			IF OP50_HORI_SERVO_ON_WRK_PICK THEN
				 SR50_Vert_servo_ctrl.Position:=OP50_VERT_SERVO_PICK_POS;
				 SR50_VERT_servo_ctrl.ABSmove_Start := TRUE;
				 OP50_AutoSeq:=100;
			 END_IF				
			   			   
	   100 : IF OP50_VERT_SERVO_ON_WRK_PICK AND NOT SR50_VERT_servo_ctrl.ABSmove_Start THEN
				 SR50_VERT_servo_ctrl.ABSmove_Start := FALSE;
				 SR50_Vert_servo_ctrl.Position:=OP50_VERT_SERVO_SFE_WRK_POS; // FEEDING SAFE-WORK POSITION TO VERTICAL SERVO
              	 OP50_AutoSeq:=110;				   
			 END_IF	   
			 
      110:  IF NOT OP50_Grip_LH_Bypass THEN
				OP50_Gripper_LH_Open:=TRUE; 
			END_IF	
			IF NOT OP50_Grip_RH_Bypass THEN
    			OP50_Gripper_RH_Open:=TRUE;
			END_IF	
			IF Gripper_Delay.Q AND NOT I50_LH_GRIP_CLSE_I1101_7 AND NOT I50_RH_GRIP_CLSE_I1110_1 THEN
				 OP50_AutoSeq:=120;
		    END_IF
    		
